(* IEC 61131-3 sources: RL_MAR/experiments/results/ablation/Ablation_random_topo_deepseek-ai_DeepSeek-V3.2_20260603_051006 (part 2) *)

(* ---- med_49.st ---- *)
FUNCTION_BLOCK SmartHVACSystem
VAR_INPUT
    TemperatureSensor : REAL; (* Temperature sensor reading *)
    HumiditySensor : REAL; (* Humidity sensor reading *)
END_VAR

VAR_OUTPUT
    HVACMode : INT := 0; (* HVAC operating mode: 0=Off, 1=Cooling, 2=Heating, 3=Ventilation *)
    HVACFanSpeed : INT := 0; (* Fan speed: 0=Off, 1=Low, 2=Medium, 3=High *)
END_VAR

VAR
    DesiredTemperature : REAL := 24.0; (* Desired temperature setting *)
    DesiredHumidity : REAL := 50.0; (* Desired humidity setting *)
    TemperatureThreshold : REAL := 1.0; (* Temperature tolerance threshold *)
    HumidityThreshold : REAL := 5.0; (* Humidity tolerance threshold *)
    AdjustedHumidity : REAL; (* Sanitized humidity input *)
    AdjustedTemperature : REAL; (* Sanitized temperature input *)
    NeedsVentilation : BOOL; (* Flag for ventilation requirement *)
    NeedsHeating : BOOL; (* Flag for heating requirement *)
    NeedsCooling : BOOL; (* Flag for cooling requirement *)
END_VAR

(* Input Sanitization *)
IF HumiditySensor < 0.0 THEN
    AdjustedHumidity := 0.0;
ELSIF HumiditySensor > 100.0 THEN
    AdjustedHumidity := 100.0;
ELSE
    AdjustedHumidity := HumiditySensor;
END_IF;

IF TemperatureSensor < -50.0 THEN
    AdjustedTemperature := -50.0;
ELSIF TemperatureSensor > 100.0 THEN
    AdjustedTemperature := 100.0;
ELSE
    AdjustedTemperature := TemperatureSensor;
END_IF;

(* Determine System Requirements *)
NeedsVentilation := AdjustedHumidity < (DesiredHumidity - HumidityThreshold);
NeedsHeating := AdjustedTemperature < (DesiredTemperature - TemperatureThreshold);
NeedsCooling := AdjustedTemperature > (DesiredTemperature + TemperatureThreshold);

(* Control Logic with Prioritization *)
IF NeedsHeating THEN
    HVACMode := 2; (* Heating mode *)
    HVACFanSpeed := 3; (* High fan speed *)
ELSIF NeedsCooling THEN
    HVACMode := 1; (* Cooling mode *)
    HVACFanSpeed := 3; (* High fan speed *)
ELSIF NeedsVentilation THEN
    HVACMode := 3; (* Ventilation mode *)
    HVACFanSpeed := 3; (* High fan speed *)
ELSE
    HVACMode := 0; (* Off mode *)
    HVACFanSpeed := 0; (* Fan off *)
END_IF;

END_FUNCTION_BLOCK

(* ---- med_50.st ---- *)
FUNCTION_BLOCK CarParkingSystem
VAR_INPUT
    NewCarSlot : INT; (* Input for new car arrival slot number *)
END_VAR
VAR_OUTPUT
    Elevator1Busy : BOOL; (* Elevator 1 status - busy or idle *)
    Elevator2Busy : BOOL; (* Elevator 2 status - busy or idle *)
    Elevator1Position : INT; (* Elevator 1 current position *)
    Elevator2Position : INT; (* Elevator 2 current position *)
END_VAR
VAR
    Elevator1Target : INT; (* Elevator 1 target floor *)
    Elevator2Target : INT; (* Elevator 2 target floor *)
    CarSlots : ARRAY[1..100] OF BOOL; (* Array to represent parking slots - TRUE if occupied *)
    CurrentSlot : INT; (* Loop counter for scanning slots *)
    bScanComplete : BOOL; (* Flag to indicate slot scanning completion *)
END_VAR

(* Initialize variables *)
IF NOT bScanComplete THEN
    Elevator1Target := 0;
    Elevator2Target := 0;
    Elevator1Position := 0;
    Elevator2Position := 0;
    Elevator1Busy := FALSE;
    Elevator2Busy := FALSE;
    CurrentSlot := 1;
    bScanComplete := TRUE;

    (* Clear all parking slots *)
    FOR CurrentSlot := 1 TO 100 DO
        CarSlots[CurrentSlot] := FALSE;
    END_FOR;
END_IF;

(* Process new car arrival *)
IF NewCarSlot >= 1 AND NewCarSlot <= 100 THEN
    IF NOT CarSlots[NewCarSlot] THEN
        CarSlots[NewCarSlot] := TRUE;

        (* Assign elevator based on slot range *)
        IF NewCarSlot <= 50 THEN
            IF NOT Elevator1Busy THEN
                Elevator1Target := NewCarSlot;
                Elevator1Busy := TRUE;
            END_IF;
        ELSE
            IF NOT Elevator2Busy THEN
                Elevator2Target := NewCarSlot;
                Elevator2Busy := TRUE;
            END_IF;
        END_IF;
    END_IF;
END_IF;

(* Elevator 1 movement logic *)
IF Elevator1Busy THEN
    IF Elevator1Position < Elevator1Target THEN
        Elevator1Position := Elevator1Position + 1;
    ELSIF Elevator1Position > Elevator1Target THEN
        Elevator1Position := Elevator1Position - 1;
    ELSE
        (* Reached target - mark as idle *)
        Elevator1Busy := FALSE;
        Elevator1Target := 0;
    END_IF;
END_IF;

(* Elevator 2 movement logic *)
IF Elevator2Busy THEN
    IF Elevator2Position < Elevator2Target THEN
        Elevator2Position := Elevator2Position + 1;
    ELSIF Elevator2Position > Elevator2Target THEN
        Elevator2Position := Elevator2Position - 1;
    ELSE
        (* Reached target - mark as idle *)
        Elevator2Busy := FALSE;
        Elevator2Target := 0;
    END_IF;
END_IF;

(* Scan for new tasks - only scan when both elevators are idle *)
IF NOT Elevator1Busy AND NOT Elevator2Busy THEN
    FOR CurrentSlot := 1 TO 100 DO
        IF CarSlots[CurrentSlot] THEN
            (* Assign to appropriate elevator *)
            IF CurrentSlot <= 50 THEN
                Elevator1Target := CurrentSlot;
                Elevator1Busy := TRUE;
                EXIT; (* Exit loop after assigning one task *)
            ELSE
                Elevator2Target := CurrentSlot;
                Elevator2Busy := TRUE;
                EXIT; (* Exit loop after assigning one task *)
            END_IF;
        END_IF;
    END_FOR;
END_IF;

END_FUNCTION_BLOCK

(* ---- med_51.st ---- *)
FUNCTION_BLOCK PizzaMakingMachine
VAR_INPUT
    StartButton : BOOL;
    StopButton : BOOL;
    DoughReadySensor : BOOL;
    ToppingsReadySensor : BOOL;
    BakingDoneSensor : BOOL;
END_VAR

VAR_OUTPUT
    DoughRollerMotor : BOOL;
    ToppingDispenser : BOOL;
    ConveyorMotor : BOOL;
    OvenHeater : BOOL;
    OvenTemperature : INT;
END_VAR

VAR
    CurrentState : INT := 0;
    NextState : INT := 0;
END_VAR

(* State Machine Execution *)
CurrentState := NextState;

CASE CurrentState OF
    0: (* IDLE STATE *)
        DoughRollerMotor := FALSE;
        ToppingDispenser := FALSE;
        ConveyorMotor := FALSE;
        OvenHeater := FALSE;
        OvenTemperature := 0;

        IF StartButton AND NOT StopButton THEN
            NextState := 1;
        ELSE
            NextState := 0;
        END_IF;

    1: (* PREPARE_DOUGH STATE *)
        DoughRollerMotor := TRUE;
        ToppingDispenser := FALSE;
        ConveyorMotor := FALSE;
        OvenHeater := FALSE;
        OvenTemperature := 0;

        IF StopButton THEN
            NextState := 0;
        ELSIF DoughReadySensor THEN
            NextState := 2;
        ELSE
            NextState := 1;
        END_IF;

    2: (* ADD_TOPPINGS STATE *)
        DoughRollerMotor := FALSE;
        ToppingDispenser := TRUE;
        ConveyorMotor := FALSE;
        OvenHeater := FALSE;
        OvenTemperature := 0;

        IF StopButton THEN
            NextState := 0;
        ELSIF ToppingsReadySensor THEN
            NextState := 3;
        ELSE
            NextState := 2;
        END_IF;

    3: (* MOVE_TO_OVEN STATE *)
        DoughRollerMotor := FALSE;
        ToppingDispenser := FALSE;
        ConveyorMotor := TRUE;
        OvenHeater := TRUE;
        OvenTemperature := 220;

        IF StopButton THEN
            NextState := 0;
        ELSIF BakingDoneSensor THEN
            NextState := 4;
        ELSE
            NextState := 3;
        END_IF;

    4: (* BAKING_COMPLETE STATE *)
        DoughRollerMotor := FALSE;
        ToppingDispenser := FALSE;
        ConveyorMotor := FALSE;
        OvenHeater := FALSE;
        OvenTemperature := 0;

        IF StopButton OR NOT StartButton THEN
            NextState := 0;
        ELSE
            NextState := 4;
        END_IF;

    ELSE
        (* Error handling: Reset to IDLE state *)
        NextState := 0;
        DoughRollerMotor := FALSE;
        ToppingDispenser := FALSE;
        ConveyorMotor := FALSE;
        OvenHeater := FALSE;
        OvenTemperature := 0;

END_CASE;

END_FUNCTION_BLOCK

(* ---- med_52.st ---- *)
FUNCTION_BLOCK TrafficManagementSystem
VAR_INPUT
    VehicleCount1 : INT;
    VehicleCount2 : INT;
    VehicleCount3 : INT;
    VehicleCount4 : INT;
END_VAR

VAR_OUTPUT
    TrafficLight1 : BOOL;  (* TRUE = Green, FALSE = Red *)
    TrafficLight2 : BOOL;
    TrafficLight3 : BOOL;
    TrafficLight4 : BOOL;
END_VAR

VAR
    tmrPair1 : TON;
    tmrPair2 : TON;
    prevCount1 : INT := 0;
    prevCount2 : INT := 0;
    prevCount3 : INT := 0;
    prevCount4 : INT := 0;
    intendedLight1 : BOOL := FALSE;
    intendedLight2 : BOOL := FALSE;
    intendedLight3 : BOOL := FALSE;
    intendedLight4 : BOOL := FALSE;
    countChangeDetected : BOOL;
END_VAR

(* Detect if any vehicle count has changed since last cycle *)
countChangeDetected := (prevCount1 <> VehicleCount1) OR
                       (prevCount2 <> VehicleCount2) OR
                       (prevCount3 <> VehicleCount3) OR
                       (prevCount4 <> VehicleCount4);

(* Timer for Pair 1 (Intersections 1 & 2) - 5 second minimum green time *)
tmrPair1(
    IN := countChangeDetected,
    PT := T#5s
);

(* Timer for Pair 2 (Intersections 3 & 4) - 5 second minimum green time *)
tmrPair2(
    IN := countChangeDetected,
    PT := T#5s
);

(* Determine intended light states for Pair 1 based on vehicle counts *)
IF VehicleCount1 > VehicleCount2 THEN
    intendedLight1 := TRUE;
    intendedLight2 := FALSE;
ELSIF VehicleCount2 > VehicleCount1 THEN
    intendedLight1 := FALSE;
    intendedLight2 := TRUE;
ELSE
    (* If counts are equal, set both to red for safety *)
    intendedLight1 := FALSE;
    intendedLight2 := FALSE;
END_IF;

(* Determine intended light states for Pair 2 based on vehicle counts *)
IF VehicleCount3 > VehicleCount4 THEN
    intendedLight3 := TRUE;
    intendedLight4 := FALSE;
ELSIF VehicleCount4 > VehicleCount3 THEN
    intendedLight3 := FALSE;
    intendedLight4 := TRUE;
ELSE
    (* If counts are equal, set both to red for safety *)
    intendedLight3 := FALSE;
    intendedLight4 := FALSE;
END_IF;

(* Apply light states with timer logic to prevent rapid toggling *)
(* Pair 1: Only update lights if timer has elapsed or no change detected *)
IF NOT tmrPair1.Q AND countChangeDetected THEN
    (* Hold current states during timer period *)
    TrafficLight1 := TrafficLight1;
    TrafficLight2 := TrafficLight2;
ELSE
    (* Apply intended states when timer elapses *)
    TrafficLight1 := intendedLight1;
    TrafficLight2 := intendedLight2;
END_IF;

(* Pair 2: Only update lights if timer has elapsed or no change detected *)
IF NOT tmrPair2.Q AND countChangeDetected THEN
    (* Hold current states during timer period *)
    TrafficLight3 := TrafficLight3;
    TrafficLight4 := TrafficLight4;
ELSE
    (* Apply intended states when timer elapses *)
    TrafficLight3 := intendedLight3;
    TrafficLight4 := intendedLight4;
END_IF;

(* Update previous counts for next cycle *)
prevCount1 := VehicleCount1;
prevCount2 := VehicleCount2;
prevCount3 := VehicleCount3;
prevCount4 := VehicleCount4;

END_FUNCTION_BLOCK

(* ---- med_53.st ---- *)
FUNCTION_BLOCK PouchMachine
VAR_INPUT
    start_machine: BOOL;
    stop_machine: BOOL;
    EmergencyStop: BOOL;
    HeatingStationReady_1: BOOL;
    HeatingStationReady_2: BOOL;
    HeatingStationReady_3: BOOL;
    HeatingStationReady_4: BOOL;
    HeatingStationReady_5: BOOL;
    HeatingStationReady_6: BOOL;
    HeatingStationReady_7: BOOL;
    HeatingStationReady_8: BOOL;
    CoolingStationReady_1: BOOL;
    CoolingStationReady_2: BOOL;
    CoolingStationReady_3: BOOL;
    CoolingStationReady_4: BOOL;
    CoolingStationReady_5: BOOL;
    CoolingStationReady_6: BOOL;
    CoolingStationReady_7: BOOL;
    CoolingStationReady_8: BOOL;
    Feeder1_TensionOK: BOOL;
    Feeder2_TensionOK: BOOL;
    HorizontalCutterReady: BOOL;
    VerticalCutterReady: BOOL;
END_VAR

VAR_OUTPUT
    machine_ready: BOOL;
    feeder_running: BOOL;
    cutter_running: BOOL;
    heating_running: BOOL;
    cooling_running: BOOL;
    Feeder1_Start: BOOL;
    Feeder2_Start: BOOL;
    HeatingStationStart_1: BOOL;
    HeatingStationStart_2: BOOL;
    HeatingStationStart_3: BOOL;
    HeatingStationStart_4: BOOL;
    HeatingStationStart_5: BOOL;
    HeatingStationStart_6: BOOL;
    HeatingStationStart_7: BOOL;
    HeatingStationStart_8: BOOL;
    CoolingStationStart_1: BOOL;
    CoolingStationStart_2: BOOL;
    CoolingStationStart_3: BOOL;
    CoolingStationStart_4: BOOL;
    CoolingStationStart_5: BOOL;
    CoolingStationStart_6: BOOL;
    CoolingStationStart_7: BOOL;
    CoolingStationStart_8: BOOL;
    HorizontalCutterStart: BOOL;
    VerticalCutterStart: BOOL;
END_VAR

VAR
    startup_complete: BOOL := FALSE;
    shutdown_complete: BOOL := FALSE;
    machine_state: INT := 0;
    startup_timer: TON;
    shutdown_timer: TON;
    heating_stations_ready: BOOL;
    cooling_stations_ready: BOOL;
    tension_established: BOOL;
    cutter_horizontal_ready: BOOL;
    cutter_vertical_ready: BOOL;
    feeder1_ready: BOOL;
    feeder2_ready: BOOL;
    start_rising_edge: R_TRIG;
    stop_rising_edge: R_TRIG;
    emergency_rising_edge: R_TRIG;
    heating_ok_array: ARRAY[1..8] OF BOOL;
    cooling_ok_array: ARRAY[1..8] OF BOOL;
END_VAR

// Edge detection for control signals
start_rising_edge(CLK := start_machine);
stop_rising_edge(CLK := stop_machine);
emergency_rising_edge(CLK := EmergencyStop);

// Initialize status arrays
heating_ok_array[1] := HeatingStationReady_1;
heating_ok_array[2] := HeatingStationReady_2;
heating_ok_array[3] := HeatingStationReady_3;
heating_ok_array[4] := HeatingStationReady_4;
heating_ok_array[5] := HeatingStationReady_5;
heating_ok_array[6] := HeatingStationReady_6;
heating_ok_array[7] := HeatingStationReady_7;
heating_ok_array[8] := HeatingStationReady_8;

cooling_ok_array[1] := CoolingStationReady_1;
cooling_ok_array[2] := CoolingStationReady_2;
cooling_ok_array[3] := CoolingStationReady_3;
cooling_ok_array[4] := CoolingStationReady_4;
cooling_ok_array[5] := CoolingStationReady_5;
cooling_ok_array[6] := CoolingStationReady_6;
cooling_ok_array[7] := CoolingStationReady_7;
cooling_ok_array[8] := CoolingStationReady_8;

// Check all heating stations are ready
heating_stations_ready := heating_ok_array[1] AND heating_ok_array[2] AND
                         heating_ok_array[3] AND heating_ok_array[4] AND
                         heating_ok_array[5] AND heating_ok_array[6] AND
                         heating_ok_array[7] AND heating_ok_array[8];

// Check all cooling stations are ready
cooling_stations_ready := cooling_ok_array[1] AND cooling_ok_array[2] AND
                         cooling_ok_array[3] AND cooling_ok_array[4] AND
                         cooling_ok_array[5] AND cooling_ok_array[6] AND
                         cooling_ok_array[7] AND cooling_ok_array[8];

// Check tension established on both feeders
tension_established := Feeder1_TensionOK AND Feeder2_TensionOK;

// Check both cutters are ready
cutter_horizontal_ready := HorizontalCutterReady;
cutter_vertical_ready := VerticalCutterReady;

// Emergency stop handling - immediate shutdown to state 0
IF EmergencyStop OR emergency_rising_edge.Q THEN
    machine_state := 0;
    startup_timer(IN := FALSE);
    shutdown_timer(IN := FALSE);
END_IF

CASE machine_state OF
    0: // Idle/Stopped state
        machine_ready := FALSE;
        feeder_running := FALSE;
        cutter_running := FALSE;
        heating_running := FALSE;
        cooling_running := FALSE;
        startup_complete := FALSE;
        shutdown_complete := TRUE;

        // Reset all output commands
        Feeder1_Start := FALSE;
        Feeder2_Start := FALSE;
        HorizontalCutterStart := FALSE;
        VerticalCutterStart := FALSE;

        HeatingStationStart_1 := FALSE;
        HeatingStationStart_2 := FALSE;
        HeatingStationStart_3 := FALSE;
        HeatingStationStart_4 := FALSE;
        HeatingStationStart_5 := FALSE;
        HeatingStationStart_6 := FALSE;
        HeatingStationStart_7 := FALSE;
        HeatingStationStart_8 := FALSE;

        CoolingStationStart_1 := FALSE;
        CoolingStationStart_2 := FALSE;
        CoolingStationStart_3 := FALSE;
        CoolingStationStart_4 := FALSE;
        CoolingStationStart_5 := FALSE;
        CoolingStationStart_6 := FALSE;
        CoolingStationStart_7 := FALSE;
        CoolingStationStart_8 := FALSE;

        IF start_rising_edge.Q AND NOT EmergencyStop THEN
            machine_state := 1;
            shutdown_complete := FALSE;
        END_IF;

    1: // Start heating stations
        heating_running := TRUE;

        // Start all heating stations
        HeatingStationStart_1 := TRUE;
        HeatingStationStart_2 := TRUE;
        HeatingStationStart_3 := TRUE;
        HeatingStationStart_4 := TRUE;
        HeatingStationStart_5 := TRUE;
        HeatingStationStart_6 := TRUE;
        HeatingStationStart_7 := TRUE;
        HeatingStationStart_8 := TRUE;

        startup_timer(IN := TRUE, PT := T#5S);
        IF startup_timer.Q AND heating_stations_ready THEN
            machine_state := 2;
            startup_timer(IN := FALSE);
        ELSIF startup_timer.Q AND NOT heating_stations_ready THEN
            // Timeout without all stations ready - go to error state
            machine_state := 99;
        END_IF;

    2: // Start cooling stations
        cooling_running := TRUE;

        // Start all cooling stations
        CoolingStationStart_1 := TRUE;
        CoolingStationStart_2 := TRUE;
        CoolingStationStart_3 := TRUE;
        CoolingStationStart_4 := TRUE;
        CoolingStationStart_5 := TRUE;
        CoolingStationStart_6 := TRUE;
        CoolingStationStart_7 := TRUE;
        CoolingStationStart_8 := TRUE;

        startup_timer(IN := TRUE, PT := T#5S);
        IF startup_timer.Q AND cooling_stations_ready THEN
            machine_state := 3;
            startup_timer(IN := FALSE);
        ELSIF startup_timer.Q AND NOT cooling_stations_ready THEN
            machine_state := 99;
        END_IF;

    3: // Start feeders and establish tension
        feeder_running := TRUE;
        Feeder1_Start := TRUE;
        Feeder2_Start := TRUE;

        startup_timer(IN := TRUE, PT := T#10S);
        IF startup_timer.Q AND tension_established THEN
            feeder1_ready := TRUE;
            feeder2_ready := TRUE;
            machine_state := 4;
            startup_timer(IN := FALSE);
        ELSIF startup_timer.Q AND NOT tension_established THEN
            machine_state := 99;
        END_IF;

    4: // Start cutters
        cutter_running := TRUE;
        HorizontalCutterStart := TRUE;
        VerticalCutterStart := TRUE;

        startup_timer(IN := TRUE, PT := T#3S);
        IF startup_timer.Q AND cutter_horizontal_ready AND cutter_vertical_ready THEN
            machine_state := 5;
            startup_timer(IN := FALSE);
        ELSIF startup_timer.Q AND NOT (cutter_horizontal_ready AND cutter_vertical_ready) THEN
            machine_state := 99;
        END_IF;

    5: // Machine ready state
        machine_ready := TRUE;
        startup_complete := TRUE;

        IF stop_rising_edge.Q OR EmergencyStop THEN
            machine_state := 10;
        END_IF;

    10: // Shutdown - stop cutters
        cutter_running := FALSE;
        HorizontalCutterStart := FALSE;
        VerticalCutterStart := FALSE;

        shutdown_timer(IN := TRUE, PT := T#3S);
        IF shutdown_timer.Q THEN
            machine_state := 11;
            shutdown_timer(IN := FALSE);
        END_IF;

    11: // Shutdown - stop feeders
        feeder_running := FALSE;
        Feeder1_Start := FALSE;
        Feeder2_Start := FALSE;

        shutdown_timer(IN := TRUE, PT := T#5S);
        IF shutdown_timer.Q THEN
            machine_state := 12;
            shutdown_timer(IN := FALSE);
        END_IF;

    12: // Shutdown - stop cooling stations
        cooling_running := FALSE;
        CoolingStationStart_1 := FALSE;
        CoolingStationStart_2 := FALSE;
        CoolingStationStart_3 := FALSE;
        CoolingStationStart_4 := FALSE;
        CoolingStationStart_5 := FALSE;
        CoolingStationStart_6 := FALSE;
        CoolingStationStart_7 := FALSE;
        CoolingStationStart_8 := FALSE;

        shutdown_timer(IN := TRUE, PT := T#5S);
        IF shutdown_timer.Q THEN
            machine_state := 13;
            shutdown_timer(IN := FALSE);
        END_IF;

    13: // Shutdown - stop heating stations
        heating_running := FALSE;
        HeatingStationStart_1 := FALSE;
        HeatingStationStart_2 := FALSE;
        HeatingStationStart_3 := FALSE;
        HeatingStationStart_4 := FALSE;
        HeatingStationStart_5 := FALSE;
        HeatingStationStart_6 := FALSE;
        HeatingStationStart_7 := FALSE;
        HeatingStationStart_8 := FALSE;

        shutdown_timer(IN := TRUE, PT := T#5S);
        IF shutdown_timer.Q THEN
            machine_state := 14;
            shutdown_timer(IN := FALSE);
        END_IF;

    14: // Shutdown complete
        machine_ready := FALSE;
        shutdown_complete := TRUE;

        IF start_rising_edge.Q AND NOT EmergencyStop THEN
            machine_state := 1;
        END_IF;

    99: // Error state
        machine_ready := FALSE;
        feeder_running := FALSE;
        cutter_running := FALSE;
        heating_running := FALSE;
        cooling_running := FALSE;

        // Stop all outputs
        Feeder1_Start := FALSE;
        Feeder2_Start := FALSE;
        HorizontalCutterStart := FALSE;
        VerticalCutterStart := FALSE;

        HeatingStationStart_1 := FALSE;
        HeatingStationStart_2 := FALSE;
        HeatingStationStart_3 := FALSE;
        HeatingStationStart_4 := FALSE;
        HeatingStationStart_5 := FALSE;
        HeatingStationStart_6 := FALSE;
        HeatingStationStart_7 := FALSE;
        HeatingStationStart_8 := FALSE;

        CoolingStationStart_1 := FALSE;
        CoolingStationStart_2 := FALSE;
        CoolingStationStart_3 := FALSE;
        CoolingStationStart_4 := FALSE;
        CoolingStationStart_5 := FALSE;
        CoolingStationStart_6 := FALSE;
        CoolingStationStart_7 := FALSE;
        CoolingStationStart_8 := FALSE;

        // Manual reset required
        IF EmergencyStop THEN
            machine_state := 0;
        END_IF;

    ELSE
        machine_state := 0;
END_CASE;
END_FUNCTION_BLOCK

(* ---- med_54.st ---- *)
FUNCTION_BLOCK FeedForwardControl
VAR_INPUT
    FlowRate1, FlowRate2: REAL; // Input flow rates of reactants
    MixRatio: REAL; // Desired mixing ratio (Reactant1:Reactant2)
END_VAR

VAR_OUTPUT
    OutFlowRate1, OutFlowRate2: REAL; // Output flow rates for reactants to maintain the mixing ratio
END_VAR

VAR
    MixedFlowRate: REAL; // Total mixed flow rate
    LimitedFlowRate1: REAL;
    LimitedFlowRate2: REAL;
    RatioSum: REAL;
END_VAR

// Limit input flow rates to valid range (0 to 100)
LimitedFlowRate1 := LIMIT(0.0, FlowRate1, 100.0);
LimitedFlowRate2 := LIMIT(0.0, FlowRate2, 100.0);

// Calculate total mixed flow rate
MixedFlowRate := LimitedFlowRate1 + LimitedFlowRate2;

// Calculate output flow rates with error handling for division by zero
RatioSum := MixRatio + 1.0;

IF RatioSum <> 0.0 THEN
    // Calculate proportional outputs based on mixing ratio
    OutFlowRate1 := MixedFlowRate * (MixRatio / RatioSum);
    OutFlowRate2 := MixedFlowRate * (1.0 / RatioSum);

    // Limit output flow rates to valid range (0 to 100)
    OutFlowRate1 := LIMIT(0.0, OutFlowRate1, 100.0);
    OutFlowRate2 := LIMIT(0.0, OutFlowRate2, 100.0);
ELSE
    // Handle division by zero case (when MixRatio = -1.0)
    OutFlowRate1 := 0.0;
    OutFlowRate2 := 0.0;
END_IF;

END_FUNCTION_BLOCK

(* ---- med_55.st ---- *)
FUNCTION_BLOCK StateMachineControl
VAR_INPUT
    request : BOOL;
    done : BOOL;
END_VAR

VAR_OUTPUT
    listen : BOOL;
END_VAR

VAR
    state : INT := 0;
END_VAR

CASE state OF
    0: (* Idle state *)
        listen := TRUE;
        IF request THEN
            state := 1;
            listen := FALSE;
        END_IF;

    1: (* Processing state *)
        listen := FALSE;
        IF done THEN
            state := 0;
        END_IF;

    ELSE
        (* Handle unexpected state values *)
        state := 0;
        listen := FALSE;
END_CASE;

END_FUNCTION_BLOCK

(* ---- med_56.st ---- *)
FUNCTION_BLOCK FB_SimpleRepeat
VAR_INPUT
    INPUT_VAR1 : INT := 2;
    INPUT_COUNTER : INT := 4;
END_VAR

VAR_OUTPUT
    OUTPUT_VAR1 : INT;
END_VAR

VAR
    COUNTER : INT;
END_VAR

// Main logic
OUTPUT_VAR1 := INPUT_VAR1;
COUNTER := INPUT_COUNTER;

REPEAT
    OUTPUT_VAR1 := OUTPUT_VAR1 * 2;
    COUNTER := COUNTER - 1;
UNTIL COUNTER = 0
END_REPEAT;

END_FUNCTION_BLOCK

(* ---- med_57.st ---- *)
FUNCTION_BLOCK FB_CourseDifferenceControl
VAR_INPUT
    KOMPASS_GRAD : INT;
    KURS : INT;
END_VAR
VAR_OUTPUT
    KURS_DIFF : INT;
END_VAR
VAR
    iDiff : INT;
END_VAR

IF KOMPASS_GRAD < 0 THEN
    KURS_DIFF := 0;
ELSE
    iDiff := KURS - KOMPASS_GRAD;

    (* Normalize the angular difference to the range [-1800, 1800] *)
    IF iDiff > 1800 THEN
        iDiff := iDiff - 3600;
    ELSIF iDiff < -1800 THEN
        iDiff := iDiff + 3600;
    END_IF;

    KURS_DIFF := iDiff;
END_IF;

END_FUNCTION_BLOCK

(* ---- med_58.st ---- *)
FUNCTION_BLOCK FB_ThresholdAccumulator
VAR_INPUT
    i : INT;
END_VAR

VAR_OUTPUT
    o : INT;
END_VAR

VAR
    s1 : INT;
END_VAR

// Main logic
s1 := 0; // Initialize s1 to 0 at the start of each call

// Process positive input values
IF i > 0 THEN
    s1 := s1 + i;
END_IF;

// Check threshold condition
IF s1 = 42 THEN
    s1 := s1 + 8000;
END_IF;

// Determine final output
IF s1 < 0 THEN
    o := 0;
ELSE
    o := s1;
END_IF;

END_FUNCTION_BLOCK

(* ---- med_59.st ---- *)
FUNCTION_BLOCK FB_ConditionalSelectAndAggregate
VAR_INPUT
    Z : INT;
END_VAR
VAR
    A_X : INT := 42;
    A_Y : INT := 333;
END_VAR
VAR_OUTPUT
    NEW_Z : INT;
END_VAR

IF A_X > Z THEN
    NEW_Z := A_Y;
ELSE
    NEW_Z := Z;
END_IF;
NEW_Z := NEW_Z + A_X + A_Y;
END_FUNCTION_BLOCK

(* ---- med_60.st ---- *)
FUNCTION_BLOCK FB_RequestHandler
VAR_INPUT
    request : BOOL;
    done : BOOL;
END_VAR

VAR_OUTPUT
    listen : BOOL;
END_VAR

VAR
    state : INT := 0;
END_VAR

CASE state OF
    0:
        listen := TRUE;
        IF request THEN
            listen := FALSE;
            state := 1;
        END_IF;

    1:
        listen := FALSE;
        IF done THEN
            listen := TRUE;
            state := 0;
        END_IF;
END_CASE;

END_FUNCTION_BLOCK

(* ---- med_61.st ---- *)
FUNCTION_BLOCK FB_Sum
VAR_INPUT
    maxValue : INT;
END_VAR
VAR_OUTPUT
    wData : WORD;
END_VAR
VAR
    II : INT;
    tempSum : DINT; // Temporary variable for summation
END_VAR

// Initialize
tempSum := 0;
wData := 0;

// Summation loop
FOR II := 0 TO maxValue DO
    tempSum := tempSum + II;
END_FOR

// Assign result with range checking
IF tempSum >= 0 AND tempSum <= 65535 THEN
    wData := WORD(tempSum);
ELSE
    wData := 0; // Handle overflow by resetting to 0
END_IF
END_FUNCTION_BLOCK

(* ---- med_62.st ---- *)
FUNCTION_BLOCK FB_PedestrianTrafficLight
VAR_INPUT
    pedBtnPress : BOOL;
END_VAR
VAR_OUTPUT
    carLightIsGreen : BOOL;
    pedLightIsGreen : BOOL;
    TimeCounter : INT;
END_VAR
VAR
    buttonPressedBefore : BOOL := FALSE;
    CurrentState : INT := 0;
    NextState : INT := 0;
    pedBtnEdge : R_TRIG;
END_VAR

// Edge detection for button press
pedBtnEdge(CLK := pedBtnPress);

// State machine execution
CASE CurrentState OF
    0: // STATE_CAR_GREEN_IDLE
        // Actions executed in this state
        carLightIsGreen := TRUE;
        pedLightIsGreen := FALSE;
        TimeCounter := 0;
        buttonPressedBefore := pedBtnPress;

        // Transition logic from this state
        IF pedBtnEdge.Q AND NOT buttonPressedBefore THEN
            NextState := 1;
        ELSE
            NextState := 0;
        END_IF;

    1: // STATE_CAR_RED_COUNTING
        // Actions executed in this state
        carLightIsGreen := FALSE;
        pedLightIsGreen := FALSE;
        TimeCounter := TimeCounter + 1;

        // Transition logic from this state
        IF TimeCounter >= 10 AND TimeCounter < 40 THEN
            NextState := 2;
        ELSIF TimeCounter >= 40 AND TimeCounter < 50 THEN
            NextState := 3;
        ELSIF TimeCounter >= 50 THEN
            NextState := 0;
        ELSE
            NextState := 1;
        END_IF;

    2: // STATE_PED_GREEN_COUNTING
        // Actions executed in this state
        carLightIsGreen := FALSE;
        pedLightIsGreen := TRUE;
        TimeCounter := TimeCounter + 1;

        // Transition logic from this state
        IF TimeCounter >= 40 AND TimeCounter < 50 THEN
            NextState := 3;
        ELSIF TimeCounter >= 50 THEN
            NextState := 0;
        ELSE
            NextState := 2;
        END_IF;

    3: // STATE_PED_RED_COUNTING
        // Actions executed in this state
        carLightIsGreen := FALSE;
        pedLightIsGreen := FALSE;
        TimeCounter := TimeCounter + 1;

        // Transition logic from this state
        IF TimeCounter >= 50 THEN
            NextState := 0;
        ELSE
            NextState := 3;
        END_IF;
END_CASE;

// State transition
CurrentState := NextState;

END_FUNCTION_BLOCK

(* ---- med_63.st ---- *)
FUNCTION MoveCarToExitGate : BOOL
VAR_INPUT
    SpaceNumber : INT;
END_VAR
// Simulate car movement to exit gate
// In a real system, this would control physical actuators
MoveCarToExitGate := TRUE; // Return TRUE when movement is complete
END_FUNCTION

FUNCTION_BLOCK Automated_Parking_Controller
VAR_INPUT
    EntryGateSensor : BOOL; (* Sensor input for entry gate *)
    ExitGateSensor : BOOL; (* Sensor input for exit gate *)
    CarDetected : BOOL; (* Sensor input for car detection *)
END_VAR
VAR_OUTPUT
    ParkingSpaceNumber : INT := 0; (* Allocated parking space number *)
    RetrievalInProgress : BOOL := FALSE; (* Flag for car retrieval in progress *)
END_VAR
VAR
    ParkingSpaces : ARRAY[1..100] OF BOOL; (* Parking space status: TRUE=Occupied, FALSE=Available *)
    i : INT; (* Loop counter *)
    AssignedSpace : INT := 0; (* Temporary storage for assigned space *)
    RetrievalComplete : BOOL := FALSE; (* Flag to track retrieval completion *)
END_VAR

// Entry Gate Management
IF EntryGateSensor AND NOT RetrievalInProgress THEN
    // Find first available parking space
    AssignedSpace := 0;
    FOR i := 1 TO 100 DO
        IF NOT ParkingSpaces[i] THEN
            AssignedSpace := i;
            EXIT;
        END_IF
    END_FOR

    // If available space found, allocate it
    IF AssignedSpace > 0 THEN
        ParkingSpaces[AssignedSpace] := TRUE;
        ParkingSpaceNumber := AssignedSpace;
    END_IF
END_IF

// Exit Gate Management
IF ExitGateSensor AND (ParkingSpaceNumber > 0) THEN
    // Mark the space as available and reset output
    ParkingSpaces[ParkingSpaceNumber] := FALSE;
    ParkingSpaceNumber := 0;
END_IF

// Car Retrieval Management
IF CarDetected AND NOT RetrievalInProgress AND (ParkingSpaceNumber > 0) THEN
    RetrievalInProgress := TRUE;
    RetrievalComplete := FALSE;
END_IF

IF RetrievalInProgress AND NOT RetrievalComplete THEN
    // Execute car movement to exit gate
    RetrievalComplete := MoveCarToExitGate(ParkingSpaceNumber);

    IF RetrievalComplete THEN
        // Mark space as available and reset
        ParkingSpaces[ParkingSpaceNumber] := FALSE;
        ParkingSpaceNumber := 0;
        RetrievalInProgress := FALSE;
    END_IF
END_IF

END_FUNCTION_BLOCK

(* ---- med_64.st ---- *)
FUNCTION_BLOCK BakeryOvenControl
VAR_INPUT
    TemperatureSensor : REAL;           (* Current oven temperature measurement *)
    HumiditySensor : REAL;              (* Current oven humidity measurement *)
    TemperatureSetpoint : REAL := 180.0; (* Desired temperature setpoint *)
    HumiditySetpoint : REAL := 60.0;    (* Desired humidity setpoint *)
    BakingTimeSetpoint : TIME := T#30m; (* Total baking duration *)
    OvenEnable : BOOL;                  (* Master enable signal for oven operation *)
    TemperatureThreshold : REAL := 2.0; (* Temperature control deadband *)
    HumidityThreshold : REAL := 5.0;    (* Humidity control deadband *)
END_VAR

VAR_OUTPUT
    HeatingElement : BOOL;              (* Control output for heating element *)
    CoolingElement : BOOL;              (* Control output for cooling element *)
    HumidityControl : BOOL;             (* Control output for humidification system *)
    DehumidityControl : BOOL;           (* Control output for dehumidification system *)
    BakingComplete : BOOL;              (* Flag indicating baking cycle completion *)
    RemainingTimeDisplay : TIME;        (* Remaining baking time for display *)
END_VAR

VAR
    RemainingTime : TIME;               (* Internal remaining time counter *)
    OneSecTimer : TON;                  (* Timer for one-second intervals *)
    OvenActive : BOOL;                  (* Internal oven active state *)
    StartBaking : BOOL;                 (* Edge detection for baking start *)
    TemperatureLowLimit : REAL;         (* Calculated temperature lower limit *)
    TemperatureHighLimit : REAL;        (* Calculated temperature upper limit *)
    HumidityLowLimit : REAL;            (* Calculated humidity lower limit *)
    HumidityHighLimit : REAL;           (* Calculated humidity upper limit *)
    PrevOvenEnable : BOOL;              (* Previous state for edge detection *)
END_VAR

(* Calculate control limits based on setpoints and thresholds *)
TemperatureLowLimit := TemperatureSetpoint - TemperatureThreshold;
TemperatureHighLimit := TemperatureSetpoint + TemperatureThreshold;
HumidityLowLimit := HumiditySetpoint - HumidityThreshold;
HumidityHighLimit := HumiditySetpoint + HumidityThreshold;

(* Edge detection for oven enable signal *)
StartBaking := OvenEnable AND NOT PrevOvenEnable;
PrevOvenEnable := OvenEnable;

(* Oven state management *)
IF StartBaking THEN
    (* Initialize baking cycle when oven is first enabled *)
    RemainingTime := BakingTimeSetpoint;
    OvenActive := TRUE;
    BakingComplete := FALSE;
ELSIF NOT OvenEnable THEN
    (* Force oven inactive when enable signal is removed *)
    OvenActive := FALSE;
    BakingComplete := FALSE;
END_IF;

(* Timer logic for one-second decrement *)
OneSecTimer(IN := OvenActive, PT := T#1s);

IF OneSecTimer.Q THEN
    (* Decrement remaining time each second *)
    IF RemainingTime > T#0s THEN
        RemainingTime := RemainingTime - T#1s;
    END_IF;

    (* Check for baking completion *)
    IF RemainingTime <= T#0s THEN
        OvenActive := FALSE;
        BakingComplete := TRUE;
    END_IF;
END_IF;

(* Update display output *)
RemainingTimeDisplay := RemainingTime;

(* Temperature control logic - evaluated every scan *)
IF OvenActive AND (RemainingTime > T#0s) THEN
    (* Heating control *)
    IF TemperatureSensor < TemperatureLowLimit THEN
        HeatingElement := TRUE;
        CoolingElement := FALSE;
    (* Cooling control *)
    ELSIF TemperatureSensor > TemperatureHighLimit THEN
        HeatingElement := FALSE;
        CoolingElement := TRUE;
    (* Within acceptable range *)
    ELSE
        HeatingElement := FALSE;
        CoolingElement := FALSE;
    END_IF;

    (* Humidity control *)
    IF HumiditySensor < HumidityLowLimit THEN
        HumidityControl := TRUE;
        DehumidityControl := FALSE;
    (* Dehumidification control *)
    ELSIF HumiditySensor > HumidityHighLimit THEN
        HumidityControl := FALSE;
        DehumidityControl := TRUE;
    (* Within acceptable range *)
    ELSE
        HumidityControl := FALSE;
        DehumidityControl := FALSE;
    END_IF;
ELSE
    (* Oven inactive or baking complete - force all outputs OFF *)
    HeatingElement := FALSE;
    CoolingElement := FALSE;
    HumidityControl := FALSE;
    DehumidityControl := FALSE;
END_IF;
END_FUNCTION_BLOCK

(* ---- med_65.st ---- *)
FUNCTION_BLOCK TheaterControl
VAR_INPUT
    StartButton : BOOL;        (* Input for starting a performance *)
    StopButton : BOOL;         (* Input for stopping a performance *)
    SceneNumber : INT;         (* Input for selecting the scene or act *)
END_VAR
VAR_OUTPUT
    LightingControl : BOOL;    (* Output for controlling lighting *)
    SoundControl : BOOL;       (* Output for controlling sound *)
    PerformanceInProgress : BOOL; (* Indicator for an ongoing performance *)
END_VAR
VAR
    CurrentState : INT := 0;   (* 0=Idle, 1=Validate Scene, 2=Performance Active *)
    NextState : INT := 0;
END_VAR

(* State machine execution *)
CurrentState := NextState;

CASE CurrentState OF
    0: (* Idle State *)
        LightingControl := FALSE;
        SoundControl := FALSE;
        PerformanceInProgress := FALSE;

        IF StopButton THEN
            NextState := 0;
        ELSIF StartButton AND NOT PerformanceInProgress THEN
            NextState := 1;
        ELSE
            NextState := 0;
        END_IF;

    1: (* Validate Scene State *)
        (* Stop button has highest priority *)
        IF StopButton THEN
            NextState := 0;
        ELSIF (SceneNumber >= 1) AND (SceneNumber <= 3) THEN
            NextState := 2;
        ELSE
            (* Invalid scene number - return to idle *)
            NextState := 0;
        END_IF;

    2: (* Performance Active State *)
        LightingControl := TRUE;
        SoundControl := TRUE;
        PerformanceInProgress := TRUE;

        IF StopButton THEN
            NextState := 0;
        ELSE
            NextState := 2;
        END_IF;

    ELSE
        (* Fallback to idle state for safety *)
        NextState := 0;
END_CASE;

END_FUNCTION_BLOCK

(* ---- med_66.st ---- *)
FUNCTION_BLOCK ElevatorControl
VAR_INPUT
    CurrentPos : INT;
    RequestedPos : INT;
    ButtonPressed : BOOL;
END_VAR

VAR_OUTPUT
    MotorMovingUp : BOOL;
    MotorMovingDown : BOOL;
    DoorIsOpen : BOOL;
END_VAR

VAR
    CurrentState : INT := 0;  (* 0=Idle, 1=MovingUp, 2=MovingDown, 3=Arrived *)
    NextState : INT := 0;
END_VAR

(* State machine implementation *)
CASE CurrentState OF
    0: (* Idle State *)
        (* State actions *)
        MotorMovingUp := FALSE;
        MotorMovingDown := FALSE;
        DoorIsOpen := TRUE;

        (* Transition logic *)
        IF ButtonPressed THEN
            IF RequestedPos > CurrentPos THEN
                NextState := 1;  (* Move up *)
            ELSIF RequestedPos < CurrentPos THEN
                NextState := 2;  (* Move down *)
            ELSE
                NextState := 3;  (* Already at requested floor *)
            END_IF;
        ELSE
            NextState := 0;  (* Remain idle *)
        END_IF;

    1: (* MovingUp State *)
        (* State actions *)
        MotorMovingUp := TRUE;
        MotorMovingDown := FALSE;
        DoorIsOpen := FALSE;

        (* Transition logic *)
        IF CurrentPos = RequestedPos THEN
            NextState := 3;  (* Arrived at target floor *)
        ELSIF RequestedPos < CurrentPos THEN
            NextState := 2;  (* Switch to moving down if new request is below *)
        ELSE
            NextState := 1;  (* Continue moving up *)
        END_IF;

    2: (* MovingDown State *)
        (* State actions *)
        MotorMovingUp := FALSE;
        MotorMovingDown := TRUE;
        DoorIsOpen := FALSE;

        (* Transition logic *)
        IF CurrentPos = RequestedPos THEN
            NextState := 3;  (* Arrived at target floor *)
        ELSIF RequestedPos > CurrentPos THEN
            NextState := 1;  (* Switch to moving up if new request is above *)
        ELSE
            NextState := 2;  (* Continue moving down *)
        END_IF;

    3: (* Arrived State *)
        (* State actions *)
        MotorMovingUp := FALSE;
        MotorMovingDown := FALSE;
        DoorIsOpen := TRUE;

        (* Transition logic *)
        IF ButtonPressed THEN
            IF RequestedPos > CurrentPos THEN
                NextState := 1;  (* Move up *)
            ELSIF RequestedPos < CurrentPos THEN
                NextState := 2;  (* Move down *)
            ELSE
                NextState := 3;  (* Stay arrived *)
            END_IF;
        ELSE
            NextState := 3;  (* Remain arrived *)
        END_IF;

END_CASE;

(* Update state for next cycle *)
CurrentState := NextState;

END_FUNCTION_BLOCK

(* ---- med_67.st ---- *)
FUNCTION_BLOCK FB_FactorialCalculator
VAR_INPUT
    X : INT;
END_VAR

VAR_OUTPUT
    FactorialResult : INT;
    FactorialGoodResult : INT;
END_VAR

VAR
    tempGoodResult : INT;
END_VAR

IF (X >= -3) AND (X <= 3) THEN
    tempGoodResult := X * X * X * X;
    FactorialGoodResult := tempGoodResult;

    IF tempGoodResult > 1 THEN
        FactorialResult := tempGoodResult * (tempGoodResult - 1);
    ELSE
        FactorialResult := tempGoodResult;
    END_IF;
ELSE
    FactorialGoodResult := 0;
    FactorialResult := 1;
END_IF;

END_FUNCTION_BLOCK

(* ---- med_68.st ---- *)
FUNCTION_BLOCK FB_SignalControl
VAR_INPUT
    Int1 : BOOL;
    Int2 : BOOL;
    Int3 : BOOL;
    Int4 : BOOL;
    Int5 : BOOL;
    Int6 : BOOL;
    Int7 : BOOL;
    Int8 : BOOL;
    IntAn1 : UINT;
    IntAn2 : UINT;
    IntAn3 : UINT;
    IntAn4 : UINT;
    IntAn5 : UINT;
    IntAn6 : UINT;
    IntAn7 : UINT;
    IntAn8 : UINT;
    Marca2 : BOOL;  // Input auxiliary control flag
END_VAR

VAR_OUTPUT
    Out1 : BOOL;
    Out2 : BOOL;
    Out3 : BOOL;
    Out4 : BOOL;
    Out5 : BOOL;
    Out6 : BOOL;
    Out7 : BOOL;
    Out8 : BOOL;
    OutAn1 : UINT;
    OutAn2 : UINT;
    OutAn3 : UINT;
    OutAn4 : UINT;
    OutAn5 : UINT;
    OutAn6 : UINT;
    OutAn7 : UINT;
    OutAn8 : UINT;
END_VAR

VAR
    Marca1 : BOOL;  // Internal flag for latching control
    Marca2_Internal : BOOL;  // Internal copy of Marca2 input for logic
END_VAR

// Store input Marca2 in internal variable to avoid overwriting input
Marca2_Internal := Marca2;

// Logic for internal flag Marca1
Marca1 := (NOT Marca2_Internal) AND (Marca1 OR Out1) AND Int1;

// Logic for internal flag Marca2 (using internal copy)
Marca2_Internal := (NOT Marca1) AND (Marca2_Internal OR Out1) AND Int1;

// Latch behavior for Out1
Out1 := (NOT Marca2_Internal) AND (Marca1 OR Out1);

// Direct Boolean pass-through
Out2 := Int2;
Out3 := Int3;
Out4 := Int4;

// Direct unsigned integer pass-through
OutAn1 := IntAn1;
OutAn2 := IntAn2;
OutAn3 := IntAn3;
OutAn4 := IntAn4;

// Conditional outputs for Out5 to Out8
Out5 := (IntAn5 > 1000) AND NOT Int5;
Out6 := (IntAn6 > 1000) AND NOT Int6;
Out7 := (IntAn7 > 1000) AND NOT Int7;
Out8 := (IntAn8 > 1000) AND NOT Int8;

// Pass-through for analog outputs OutAn5 to OutAn8
OutAn5 := IntAn5;
OutAn6 := IntAn6;
OutAn7 := IntAn7;
OutAn8 := IntAn8;

END_FUNCTION_BLOCK

(* ---- med_69.st ---- *)
FUNCTION_BLOCK FB_ValueOut
VAR_INPUT
    valueIn : INT;
    conf : UINT;
END_VAR

VAR_OUTPUT
    ValueOut : INT;
END_VAR

VAR
    tempValue : INT;
END_VAR

METHOD ProcessValue : INT
VAR_INPUT
    inValue : INT;
    inConf : UINT;
END_VAR
VAR
    result : INT;
END_VAR

    result := 0;

    CASE inConf OF
        1, 2:
            IF inValue <> 0 THEN
                result := inValue / 10;
            ELSE
                result := 0;
            END_IF;

        3:
            CASE inValue OF
                0:   result := 0;
                300: result := 163;
                600: result := 331;
            ELSE
                result := 0;
            END_CASE;

        6, 7:
            IF inValue = 100 THEN
                result := 319;
            ELSE
                result := 0;
            END_IF;

    ELSE
        result := 0;
    END_CASE;

    // Ensure non-negative result
    IF result < 0 THEN
        result := 0;
    END_IF;

    ProcessValue := result;
END_METHOD

// Main execution
ValueOut := ProcessValue(valueIn := valueIn, inConf := conf);
END_FUNCTION_BLOCK

(* ---- med_70.st ---- *)
FUNCTION_BLOCK EggIncubatorControl
VAR_INPUT
    StartButton : BOOL;           (* Momentary button to start incubation *)
    StopButton : BOOL;            (* Momentary button to stop incubation *)
    TemperatureSensor : REAL;     (* Current temperature in °C *)
    HumiditySensor : REAL;        (* Current humidity in % *)
END_VAR
VAR_OUTPUT
    HeatingElement : BOOL;        (* Controls heating element *)
    Humidifier : BOOL;            (* Controls humidifier *)
    EggTurningMotor : BOOL;       (* Controls egg turning motor *)
    IncubationInProgress : BOOL;  (* Indicates if incubation is active *)
END_VAR
VAR
    TargetTemperature : REAL;     (* Target temperature setpoint *)
    TargetHumidity : REAL;        (* Target humidity setpoint *)
    TurnIntervalSeconds : INT;    (* Time interval for egg turning *)
    TurnTimerSeconds : INT;       (* Timer for egg turning cycle *)
    TurnMotorState : BOOL;        (* Internal state for motor toggle *)
END_VAR

(* Initialization of parameters *)
TargetTemperature := 37.5;
TargetHumidity := 50.0;
TurnIntervalSeconds := 3600;

(* Main control logic *)
IF StopButton THEN
    (* Emergency/Manual Stop: Reset all outputs and timers *)
    IncubationInProgress := FALSE;
    HeatingElement := FALSE;
    Humidifier := FALSE;
    EggTurningMotor := FALSE;
    TurnTimerSeconds := 0;
    TurnMotorState := FALSE;
ELSIF StartButton AND NOT IncubationInProgress THEN
    (* Start incubation process *)
    IncubationInProgress := TRUE;
    TurnTimerSeconds := 0;
    TurnMotorState := FALSE;
END_IF;

(* Temperature Control - only active when incubation is in progress *)
IF IncubationInProgress THEN
    HeatingElement := TemperatureSensor < TargetTemperature;
ELSE
    HeatingElement := FALSE;
END_IF;

(* Humidity Control - only active when incubation is in progress *)
IF IncubationInProgress THEN
    Humidifier := HumiditySensor < TargetHumidity;
ELSE
    Humidifier := FALSE;
END_IF;

(* Egg Turning Cycle - only active when incubation is in progress *)
IF IncubationInProgress THEN
    (* Increment timer each scan cycle *)
    TurnTimerSeconds := TurnTimerSeconds + 1;

    (* Check if turning interval has been reached *)
    IF TurnTimerSeconds >= TurnIntervalSeconds THEN
        (* Toggle motor state and reset timer *)
        TurnMotorState := NOT TurnMotorState;
        TurnTimerSeconds := 0;
    END_IF;

    (* Output motor state *)
    EggTurningMotor := TurnMotorState;
ELSE
    (* When not in progress, ensure motor is off *)
    EggTurningMotor := FALSE;
    TurnTimerSeconds := 0;
    TurnMotorState := FALSE;
END_IF;

END_FUNCTION_BLOCK

(* ---- med_71.st ---- *)
FUNCTION_BLOCK FB_Fibonacci_Calculator
VAR_INPUT
    N : DINT := 5;
END_VAR
VAR_OUTPUT
    O : DINT := 1;
END_VAR
VAR
    F1 : DINT := 1;
    F2 : DINT := 1;
    CNT : DINT := 2;
    MaxValue : DINT := 32767;
    Temp : DINT;
END_VAR

// Handle edge cases for N <= 2
IF N <= 2 THEN
    O := 1;
    RETURN;
END_IF

// Initialize for N > 2
F1 := 1;
F2 := 1;
CNT := 2;

// Calculate Fibonacci sequence with saturation
WHILE CNT < N DO
    // Check for overflow before calculation
    IF (F1 > (MaxValue - F2)) THEN
        O := MaxValue;
        RETURN;
    END_IF

    Temp := F1 + F2;
    F1 := F2;
    F2 := Temp;
    CNT := CNT + 1;
END_WHILE

O := F2;
END_FUNCTION_BLOCK

PROGRAM Main
VAR
    FibonacciCalc : FB_Fibonacci_Calculator;
    InputValue : DINT := 5;
    Result : DINT;
END_VAR

FibonacciCalc(N := InputValue);
Result := FibonacciCalc.O;
END_PROGRAM

(* ---- med_72.st ---- *)
FUNCTION_BLOCK DigitalSignageManagement
VAR_INPUT
    DisplayLocations : ARRAY[1..10] OF BOOL;    (* Display active status at each location *)
    ContentSource : ARRAY[1..10] OF INT;        (* Requested content for each location *)
END_VAR
VAR_OUTPUT
    CurrentContent : ARRAY[1..10] OF INT;       (* Current displayed content: 1=News, 2=Weather, 3=Promo, 0=None *)
END_VAR
VAR
    i : INT;                                    (* Loop counter *)
END_VAR

(* Main logic: Update content for all locations immediately *)
FOR i := 1 TO 10 DO
    IF DisplayLocations[i] THEN
        (* Display is active - check content source *)
        CASE ContentSource[i] OF
            1: CurrentContent[i] := 1;          (* News *)
            2: CurrentContent[i] := 2;          (* Weather *)
            3: CurrentContent[i] := 3;          (* Promotional Content *)
        ELSE
            CurrentContent[i] := 0;             (* Invalid content code or 0 *)
        END_CASE;
    ELSE
        (* Display is inactive - show no content *)
        CurrentContent[i] := 0;
    END_IF;
END_FOR;

END_FUNCTION_BLOCK

(* ---- med_73.st ---- *)
FUNCTION_BLOCK RoboticWeldingSystem
VAR_INPUT
    RobotArm1Ready : BOOL;    (* Input for robot arm 1 ready status *)
    RobotArm2Ready : BOOL;    (* Input for robot arm 2 ready status *)
    WeldingGunReady : BOOL;   (* Input for welding gun ready status *)
    StartButton : BOOL;       (* Input for start button press *)
    StopButton : BOOL;        (* Input for stop button press *)
END_VAR

VAR_OUTPUT
    WeldingTrigger : BOOL;    (* Output to trigger welding *)
    WeldingComplete : BOOL;   (* Output indicating welding completion *)
END_VAR

VAR
    CurrentState : INT;       (* 0=Idle, 1=Welding, 2=Stopped *)
    AllReady : BOOL;          (* Combined ready status *)
    ReadyLost : BOOL;         (* Flag for lost readiness during welding *)
END_VAR

(* Calculate combined conditions *)
AllReady := RobotArm1Ready AND RobotArm2Ready AND WeldingGunReady;
ReadyLost := NOT AllReady;

(* State machine implementation *)
CASE CurrentState OF
    0: (* Idle State *)
        WeldingTrigger := FALSE;
        WeldingComplete := TRUE;

        IF StopButton THEN
            CurrentState := 2;  (* Go to Stopped state *)
        ELSIF StartButton AND AllReady THEN
            CurrentState := 1;  (* Go to Welding state *)
        ELSE
            CurrentState := 0;  (* Remain in Idle *)
        END_IF;

    1: (* Welding State *)
        WeldingTrigger := TRUE;
        WeldingComplete := FALSE;

        IF StopButton THEN
            CurrentState := 2;  (* Go to Stopped state *)
        ELSIF ReadyLost THEN
            CurrentState := 0;  (* Go to Idle state *)
        ELSE
            CurrentState := 1;  (* Remain in Welding *)
        END_IF;

    2: (* Stopped State *)
        WeldingTrigger := FALSE;
        WeldingComplete := TRUE;

        IF NOT StopButton THEN
            CurrentState := 0;  (* Go to Idle state *)
        ELSE
            CurrentState := 2;  (* Remain in Stopped *)
        END_IF;

    ELSE
        (* Default to Idle state if invalid state *)
        CurrentState := 0;
        WeldingTrigger := FALSE;
        WeldingComplete := TRUE;
END_CASE;

END_FUNCTION_BLOCK

(* ---- med_74.st ---- *)
FUNCTION_BLOCK TrafficManagementSystem
VAR_INPUT
    VehicleCount1 : INT; (* Input for vehicle count at intersection 1 *)
    VehicleCount2 : INT; (* Input for vehicle count at intersection 2 *)
    VehicleCount3 : INT; (* Input for vehicle count at intersection 3 *)
    VehicleCount4 : INT; (* Input for vehicle count at intersection 4 *)
END_VAR
VAR_OUTPUT
    TrafficLight1 : BOOL; (* Output for traffic light at intersection 1 *)
    TrafficLight2 : BOOL; (* Output for traffic light at intersection 2 *)
    TrafficLight3 : BOOL; (* Output for traffic light at intersection 3 *)
    TrafficLight4 : BOOL; (* Output for traffic light at intersection 4 *)
END_VAR

(* Main logic *)
TrafficLight1 := (VehicleCount1 > VehicleCount2);
TrafficLight2 := NOT TrafficLight1;
TrafficLight3 := (VehicleCount3 > VehicleCount4);
TrafficLight4 := NOT TrafficLight3;

END_FUNCTION_BLOCK

(* ---- med_75.st ---- *)
FUNCTION_BLOCK HomeBrewingSystem
VAR_INPUT
    TemperatureSensor : REAL;      (* Current temperature in °C *)
    WaterFlowSensor : REAL;        (* Current water flow in L/min *)
    BrewingStartTime : TIME;       (* Start time of brewing process *)
    BrewingDuration : TIME;        (* Total duration of brewing process *)
END_VAR
VAR_OUTPUT
    HeatingElement : BOOL;         (* Control signal for heating element *)
    AgitationMotor : BOOL;         (* Control signal for agitation motor *)
    HopsDispenser : BOOL;          (* Control signal for hops dispenser *)
    FermentationTank : BOOL;       (* Control signal for fermentation tank transfer *)
END_VAR
VAR
    CurrentTime : TIME;            (* Current system time *)
    ElapsedTime : TIME;            (* Time elapsed since brewing start *)
    ProcessActive : BOOL;          (* Flag indicating if brewing process is active *)
END_VAR

(* Calculate current time and elapsed brewing time *)
CurrentTime := TIME();
ElapsedTime := CurrentTime - BrewingStartTime;

(* Determine if brewing process is within scheduled duration *)
ProcessActive := (ElapsedTime >= T#0s) AND (ElapsedTime <= BrewingDuration);

(* Temperature control: Maintain 65°C *)
IF TemperatureSensor < 65.0 THEN
    HeatingElement := TRUE;
ELSE
    HeatingElement := FALSE;
END_IF;

(* Agitation motor control based on water flow *)
IF WaterFlowSensor > 0.5 THEN
    AgitationMotor := TRUE;
ELSE
    AgitationMotor := FALSE;
END_IF;

(* Hops dispensing after 5 hours, only during active brewing process *)
IF ProcessActive AND (ElapsedTime >= T#5h) THEN
    HopsDispenser := TRUE;
ELSE
    HopsDispenser := FALSE;
END_IF;

(* Fermentation tank transfer after 48 hours, only during active brewing process *)
IF ProcessActive AND (ElapsedTime >= T#48h) THEN
    FermentationTank := TRUE;
ELSE
    FermentationTank := FALSE;
END_IF;

END_FUNCTION_BLOCK

(* ---- med_76.st ---- *)
FUNCTION_BLOCK MultimediaArtInstallationControl
VAR_INPUT
    MotionSensor : BOOL;           (* Motion detection input *)
    AudioTrack : BOOL;             (* Selected audio track *)
    VisualContent : BOOL;          (* Selected visual content *)
    CycleTime : TIME := T#1S;      (* Cycle time for timer increment *)
    MaxDuration : TIME := T#300S;  (* Maximum activation duration *)
END_VAR
VAR_OUTPUT
    LightingControl : BOOL;        (* Lighting control output *)
    AudioControl : BOOL;           (* Audio playback control *)
    VisualControl : BOOL;          (* Visual display control *)
    ActivationTime : TIME;         (* Current activation duration *)
    SystemActive : BOOL;           (* Overall system status *)
END_VAR
VAR
    ActivationTimer : TON;         (* Timer for activation duration *)
    ElapsedTime : TIME;            (* Elapsed activation time *)
    PreviousMotion : BOOL;         (* Previous motion state for edge detection *)
    MotionDetected : BOOL;         (* Rising edge detected motion *)
END_VAR

(* Initialize timer *)
ActivationTimer(IN := MotionSensor, PT := MaxDuration);

(* Detect rising edge of motion *)
MotionDetected := MotionSensor AND NOT PreviousMotion;
PreviousMotion := MotionSensor;

(* Control multimedia elements based on motion detection *)
IF MotionSensor THEN
    (* Activate all elements when motion is detected *)
    LightingControl := TRUE;
    AudioControl := AudioTrack;    (* Only activate if audio track is selected *)
    VisualControl := VisualContent; (* Only activate if visual content is selected *)
    SystemActive := TRUE;

    (* Update elapsed time while motion is detected *)
    IF ActivationTimer.Q THEN
        (* Timer has reached maximum duration *)
        ElapsedTime := MaxDuration;
    ELSE
        (* Calculate elapsed time based on timer's ET output *)
        ElapsedTime := ActivationTimer.ET;
    END_IF;
ELSE
    (* Deactivate all elements when no motion is detected *)
    LightingControl := FALSE;
    AudioControl := FALSE;
    VisualControl := FALSE;
    SystemActive := FALSE;

    (* Reset elapsed time *)
    ElapsedTime := T#0S;

    (* Reset the timer *)
    ActivationTimer(IN := FALSE);
END_IF;

(* Assign output *)
ActivationTime := ElapsedTime;

(* Safety protocol: Power usage monitoring *)
(* This is a placeholder for actual power monitoring logic *)
(* In a real system, you would implement:
   - Current monitoring
   - Temperature sensing
   - Emergency shutdown procedures *)

END_FUNCTION_BLOCK

(* ---- med_77.st ---- *)
FUNCTION_BLOCK OutdoorLEDLightingControl
VAR_INPUT
    AmbientLight : REAL;    (* Ambient light sensor input in Lux *)
    MotionSensor : BOOL;    (* Motion sensor input (TRUE = motion detected) *)
    EnergySaving : BOOL;    (* Energy saving mode switch (TRUE = energy saving ON) *)
END_VAR

VAR_OUTPUT
    Light : BOOL;           (* LED lighting control output (TRUE = lights ON) *)
    EnergyMode : BOOL;      (* Energy saving mode status output *)
END_VAR

(* Main control logic *)
IF MotionSensor THEN
    (* Motion Detection Override: Lights ON, EnergyMode reflects input *)
    Light := TRUE;
ELSE
    (* No motion detected - Ambient Light and Energy Saving Control *)
    IF (AmbientLight < 50.0) AND NOT EnergySaving THEN
        Light := TRUE;
    ELSE
        Light := FALSE;
    END_IF;
END_IF;

(* Energy Mode Status always reflects EnergySaving input *)
EnergyMode := EnergySaving;

END_FUNCTION_BLOCK

(* ---- med_78.st ---- *)
FUNCTION_BLOCK RetractableRoofControl
VAR_INPUT
    RainSensor : BOOL;           (* TRUE if rain is detected *)
    WindSensor : BOOL;           (* TRUE if strong wind is detected *)
    TemperatureSensor : REAL;    (* Current temperature in degrees *)
END_VAR
VAR_OUTPUT
    RoofMotor : BOOL;            (* TRUE = close roof, FALSE = open roof *)
END_VAR

(* Main control logic *)
IF RainSensor AND WindSensor THEN
    (* Highest priority: both rain and strong wind *)
    RoofMotor := TRUE;
ELSIF RainSensor THEN
    (* Second priority: rain only *)
    RoofMotor := TRUE;
ELSIF TemperatureSensor < 20.0 THEN
    (* Third priority: low temperature *)
    RoofMotor := TRUE;
ELSE
    (* Normal conditions: open roof *)
    RoofMotor := FALSE;
END_IF;

END_FUNCTION_BLOCK

(* ---- med_79.st ---- *)
FUNCTION_BLOCK CapsuleFillingMachineControl
VAR_INPUT
    CapsuleWeight : REAL;          (* Current capsule weight *)
    TargetWeight : REAL;           (* Target weight to achieve *)
    CapsuleInPosition : BOOL;      (* Capsule position sensor *)
    HopperEmpty : BOOL;            (* Hopper empty sensor *)
END_VAR

VAR_OUTPUT
    FeederMotor : BOOL;            (* Feeder motor control *)
    FillingMotor : BOOL;           (* Filling motor control *)
    ConveyorMotor : BOOL;          (* Conveyor motor control *)
    FillingInProgress : BOOL;      (* Filling status *)
    ErrorCode : INT;               (* Error code: 0=OK, 1=Capsule timeout, 2=Filling timeout *)
END_VAR

VAR
    // State machine
    CurrentState : INT;            (* 0=IDLE, 1=CONVEYING, 2=FILLING, 3=CONVEYING_OUT *)

    // Timers
    ConveyorTimer : TON;
    FillingTimer : TON;
    ConveyOutTimer : TON;

    // Timing parameters
    ConveyorTime : TIME := T#2S;   (* Time to convey capsule to filling station *)
    MaxFillingTime : TIME := T#10S; (* Maximum allowed filling time *)
    ConveyOutTime : TIME := T#1S;  (* Time to convey filled capsule out *)

    // Control variables
    WeightTolerance : REAL := 0.01; (* 1% tolerance for weight comparison *)
    TargetReached : BOOL;
    FillingStarted : BOOL;

    // Error handling
    CapsuleTimeoutError : BOOL;
    FillingTimeoutError : BOOL;

    // PID-like control variables (simplified proportional control)
    Kp : REAL := 0.8;              (* Proportional gain *)
    PreviousError : REAL;
    ControlOutput : REAL;
    MinMotorSpeed : REAL := 0.1;   (* Minimum motor speed to prevent stalling *)
END_VAR

// Initialize timers
ConveyorTimer(IN:=FALSE, PT:=ConveyorTime);
FillingTimer(IN:=FALSE, PT:=MaxFillingTime);
ConveyOutTimer(IN:=FALSE, PT:=ConveyOutTime);

// Safety Check: Hopper Empty
IF HopperEmpty THEN
    FeederMotor := FALSE;
    FillingMotor := FALSE;
    ConveyorMotor := FALSE;
    FillingInProgress := FALSE;
    CurrentState := 0;  // Return to IDLE state
    ErrorCode := 0;
    RETURN;
END_IF

// Weight Validation: Initial Check
IF CapsuleWeight >= TargetWeight THEN
    FeederMotor := FALSE;
    FillingMotor := FALSE;
    ConveyorMotor := FALSE;
    FillingInProgress := FALSE;
    CurrentState := 0;  // Return to IDLE state
    ErrorCode := 0;
    RETURN;
END_IF

// Calculate if target weight is reached (within tolerance)
TargetReached := (CapsuleWeight >= TargetWeight * (1 - WeightTolerance))
                 AND (CapsuleWeight <= TargetWeight * (1 + WeightTolerance));

// State Machine Implementation
CASE CurrentState OF
    0: (* IDLE State *)
        FeederMotor := FALSE;
        FillingMotor := FALSE;
        ConveyorMotor := FALSE;
        FillingInProgress := FALSE;
        ErrorCode := 0;

        IF CapsuleInPosition THEN
            CurrentState := 1;  // Move to CONVEYING state
            ConveyorTimer(IN:=TRUE);  // Start conveyor timer
        END_IF

    1: (* CONVEYING State *)
        ConveyorMotor := TRUE;
        FillingInProgress := FALSE;

        ConveyorTimer(IN:=TRUE);  // Keep timer running

        IF ConveyorTimer.Q THEN
            // Conveyor timed out without capsule detection
            ConveyorMotor := FALSE;
            CapsuleTimeoutError := TRUE;
            ErrorCode := 1;
            CurrentState := 0;  // Return to IDLE
        ELSIF CapsuleInPosition THEN
            // Capsule successfully conveyed to filling station
            ConveyorTimer(IN:=FALSE);  // Reset timer
            CurrentState := 2;  // Move to FILLING state
            FillingTimer(IN:=TRUE);  // Start filling timer
            FillingStarted := TRUE;
            PreviousError := TargetWeight - CapsuleWeight;  // Initialize error for control
        END_IF

    2: (* FILLING State *)
        ConveyorMotor := FALSE;
        FillingInProgress := TRUE;

        // Simplified proportional control for filling motor
        IF NOT TargetReached AND NOT FillingTimer.Q THEN
            // Calculate error
            VAR
                Error : REAL;
            END_VAR

            Error := TargetWeight - CapsuleWeight;

            // Proportional control with minimum speed
            ControlOutput := Kp * Error;
            IF ControlOutput < MinMotorSpeed THEN
                ControlOutput := MinMotorSpeed;
            ELSIF ControlOutput > 1.0 THEN
                ControlOutput := 1.0;
            END_IF

            // Convert control output to motor command (simplified)
            FillingMotor := TRUE;
            FeederMotor := TRUE;  // Activate feeder to supply material

            PreviousError := Error;
        ELSE
            FillingMotor := FALSE;
            FeederMotor := FALSE;

            IF TargetReached THEN
                // Successful filling
                FillingTimer(IN:=FALSE);  // Reset timer
                CurrentState := 3;  // Move to CONVEYING_OUT state
                ConveyOutTimer(IN:=TRUE);  // Start convey out timer
            ELSIF FillingTimer.Q THEN
                // Filling timeout
                FillingTimeoutError := TRUE;
                ErrorCode := 2;
                CurrentState := 0;  // Return to IDLE
            END_IF
        END_IF

    3: (* CONVEYING_OUT State *)
        FillingMotor := FALSE;
        FeederMotor := FALSE;
        ConveyorMotor := TRUE;
        FillingInProgress := FALSE;

        ConveyOutTimer(IN:=TRUE);  // Keep timer running

        IF ConveyOutTimer.Q THEN
            // Finished conveying out
            ConveyorMotor := FALSE;
            ConveyOutTimer(IN:=FALSE);  // Reset timer
            CurrentState := 0;  // Return to IDLE
        END_IF

END_CASE;

// Reset error flags when returning to IDLE state
IF CurrentState = 0 THEN
    CapsuleTimeoutError := FALSE;
    FillingTimeoutError := FALSE;
END_IF

END_FUNCTION_BLOCK

(* ---- med_80.st ---- *)
FUNCTION_BLOCK DoughMixerControl
VAR_INPUT
    IngredientsDetected : BOOL; (* Input for detecting the presence of ingredients *)
END_VAR

VAR_OUTPUT
    MixingInProgress : BOOL; (* Output for controlling the mixing process - on/off *)
END_VAR

VAR
    MixingTimeElapsed : TIME; (* Timer to track the mixing time *)
    MixingTimeLimit : TIME := T#5S; (* Mixing time limit - 5 seconds *)
    IngredientsDetectedPrev : BOOL; (* Previous state for edge detection *)
    StartTime : TIME; (* Stores the system time when mixing starts *)
    SystemTime : TIME; (* Current system time *)
END_VAR

(* Main logic *)
SystemTime := TIME(); (* Get current system time *)

(* Rising edge detection for IngredientsDetected *)
IF IngredientsDetected AND NOT IngredientsDetectedPrev THEN
    (* Start mixing cycle *)
    MixingInProgress := TRUE;
    StartTime := SystemTime; (* Record start time *)
    MixingTimeElapsed := T#0S; (* Reset elapsed time *)
END_IF;

(* Update previous state for next cycle *)
IngredientsDetectedPrev := IngredientsDetected;

(* Stop conditions *)
IF NOT IngredientsDetected THEN
    (* Stop if ingredients are no longer detected *)
    MixingInProgress := FALSE;
ELSIF MixingInProgress THEN
    (* Calculate elapsed time while mixing *)
    MixingTimeElapsed := SystemTime - StartTime;

    (* Stop if time limit is reached *)
    IF MixingTimeElapsed >= MixingTimeLimit THEN
        MixingInProgress := FALSE;
    END_IF;
END_IF;

(* Ensure timer doesn't increment when not mixing *)
IF NOT MixingInProgress THEN
    MixingTimeElapsed := MixingTimeElapsed; (* Hold current value *)
END_IF;
END_FUNCTION_BLOCK

(* ---- med_81.st ---- *)
FUNCTION_BLOCK SolarPanelTracking
VAR
    PanelAngle : REAL; (* Output for adjusting the solar panel angle *)
    SunriseTime : TIME := T#6H; (* Set the time for sunrise (6:00 AM) *)
    SunsetTime : TIME := T#18H; (* Set the time for sunset (6:00 PM) *)
    NoonTime : TIME := T#12H; (* Set the time for solar noon (12:00 PM) *)
    MorningAngle : REAL := 30.0; (* Set the morning angle for panels *)
    NoonAngle : REAL := 60.0; (* Set the noon angle for panels *)
    EveningAngle : REAL := 30.0; (* Set the evening angle for panels *)
END_VAR
VAR_INPUT
    CurrentTime : TIME;
    SolarIntensity : REAL;
END_VAR

(* Main execution logic *)
IF SolarIntensity >= 90.0 THEN
    (* Solar intensity override - maximum energy capture *)
    PanelAngle := NoonAngle;
ELSE
    (* Time-based tracking logic *)
    IF (CurrentTime < SunriseTime) OR (CurrentTime >= SunsetTime) THEN
        (* Nighttime - panel horizontal *)
        PanelAngle := 0.0;
    ELSIF (CurrentTime >= SunriseTime) AND (CurrentTime < NoonTime) THEN
        (* Morning period *)
        PanelAngle := MorningAngle;
    ELSE
        (* Afternoon/Evening period (NoonTime <= CurrentTime < SunsetTime) *)
        PanelAngle := EveningAngle;
    END_IF;
END_IF;

END_FUNCTION_BLOCK

(* ---- med_82.st ---- *)
FUNCTION_BLOCK PetFeederControl
VAR_INPUT
    CurrentTime : TIME; (* Current system time input *)
END_VAR

VAR_OUTPUT
    FoodDispense : BOOL; (* Food dispenser control signal *)
END_VAR

VAR
    FeedTime1 : TIME := T#8H0M0S; (* First feeding time - 8:00 AM *)
    FeedTime2 : TIME := T#12H0M0S; (* Second feeding time - 12:00 PM *)
    FeedTime3 : TIME := T#18H0M0S; (* Third feeding time - 6:00 PM *)
    FoodAmount : INT := 50; (* Amount of food to dispense in grams - currently unused *)
END_VAR

(* Main dispensing logic *)
FoodDispense := FALSE; (* Default state *)

(* Check if current time is within 30 seconds after FeedTime1 *)
IF (CurrentTime >= FeedTime1) AND (CurrentTime < FeedTime1 + T#30S) THEN
    FoodDispense := TRUE;
END_IF;

(* Check if current time is within 30 seconds after FeedTime2 *)
IF (CurrentTime >= FeedTime2) AND (CurrentTime < FeedTime2 + T#30S) THEN
    FoodDispense := TRUE;
END_IF;

(* Check if current time is within 30 seconds after FeedTime3 *)
IF (CurrentTime >= FeedTime3) AND (CurrentTime < FeedTime3 + T#30S) THEN
    FoodDispense := TRUE;
END_IF;

END_FUNCTION_BLOCK

(* ---- med_83.st ---- *)
FUNCTION_BLOCK AmusementRideControl
VAR_INPUT
    StartButton : BOOL;        (* Start button input *)
    StopButton : BOOL;         (* Emergency stop button input *)
    SpeedSensor : REAL;        (* Speed sensor input (RPM) *)
    SafetySensor : BOOL;       (* Safety sensor status *)
    ResetButton : BOOL;        (* Manual reset button - required after safety trips *)
END_VAR
VAR_OUTPUT
    MotorOn : BOOL := FALSE;   (* Motor control output *)
    BrakeOn : BOOL := TRUE;    (* Brake control output - default fail-safe *)
END_VAR
VAR
    SpeedLimit : REAL := 60.0; (* Maximum allowed speed in RPM *)
    SafetyTrip : BOOL := FALSE;(* Latched safety sensor trip *)
    OverspeedTrip : BOOL := FALSE; (* Latched overspeed trip *)
    EmergencyStopActive : BOOL := FALSE; (* Emergency stop status *)
END_VAR

(* Main safety logic - executed each scan cycle *)
(* HIGHEST PRIORITY: Emergency Stop Handling *)
IF StopButton THEN
    EmergencyStopActive := TRUE;
    MotorOn := FALSE;
    BrakeOn := TRUE;
    (* Emergency stop overrides all other logic *)
    RETURN; (* Exit logic execution for this scan *)
ELSE
    EmergencyStopActive := FALSE;
END_IF;

(* Check for safety violations during operation *)
IF MotorOn THEN
    (* Continuous monitoring while motor is running *)
    IF SpeedSensor > SpeedLimit THEN
        OverspeedTrip := TRUE;
    END_IF;

    IF NOT SafetySensor THEN
        SafetyTrip := TRUE;
    END_IF;
END_IF;

(* Safety Trip Response - Second Highest Priority *)
IF OverspeedTrip OR SafetyTrip THEN
    MotorOn := FALSE;
    BrakeOn := TRUE;
    (* Safety trips require manual reset - do not auto-restart *)
    RETURN; (* Exit logic execution for this scan *)
END_IF;

(* Manual Reset Logic *)
IF ResetButton AND NOT MotorOn THEN
    OverspeedTrip := FALSE;
    SafetyTrip := FALSE;
END_IF;

(* START CONDITION: All conditions must be met simultaneously *)
(* Requires manual reset after any trip *)
IF StartButton
   AND NOT StopButton
   AND (SpeedSensor <= SpeedLimit)
   AND SafetySensor
   AND NOT OverspeedTrip
   AND NOT SafetyTrip
   AND NOT EmergencyStopActive THEN
    (* All start conditions satisfied *)
    MotorOn := TRUE;
    BrakeOn := FALSE;
ELSE
    (* Default fail-safe state *)
    MotorOn := FALSE;
    BrakeOn := TRUE;
END_IF;

END_FUNCTION_BLOCK

(* ---- med_84.st ---- *)
FUNCTION_BLOCK ParcelSortingSystem
VAR_INPUT
    ParcelSizeSensor : REAL;           (* Sensor input for parcel size in mm *)
    DestinationCodeSensor : INT;       (* Destination code: 1=Location A, 2=Location B *)
END_VAR
VAR_OUTPUT
    ConveyorBeltMotor : BOOL;          (* Output for conveyor belt motor: TRUE=On, FALSE=Off *)
    SortingGate1 : BOOL;               (* Output for sorting gate 1: TRUE=Open, FALSE=Closed *)
    SortingGate2 : BOOL;               (* Output for sorting gate 2: TRUE=Open, FALSE=Closed *)
END_VAR
VAR
    SizeThreshold : REAL := 100.0;     (* Threshold to distinguish large vs small parcels *)
    IsLargeParcel : BOOL;              (* Flag indicating parcel is large (>= threshold) *)
    IsSmallParcel : BOOL;              (* Flag indicating parcel is small (< threshold) *)
    IsValidDestination : BOOL;         (* Flag indicating destination code is valid *)
    IsValidSize : BOOL;                (* Flag indicating parcel size is valid *)
END_VAR

(* Initialize outputs to safe default states - all off/closed *)
ConveyorBeltMotor := FALSE;
SortingGate1 := FALSE;
SortingGate2 := FALSE;

(* Validate sensor inputs *)
IsValidSize := (ParcelSizeSensor > 0.0);                    (* Valid size must be positive *)
IsValidDestination := (DestinationCodeSensor = 1) OR (DestinationCodeSensor = 2);  (* Only codes 1 or 2 are valid *)

(* Determine parcel size category based on threshold *)
IsLargeParcel := (ParcelSizeSensor >= SizeThreshold) AND IsValidSize;
IsSmallParcel := (ParcelSizeSensor < SizeThreshold) AND (ParcelSizeSensor > 0.0) AND IsValidSize;

(* Main sorting logic - only execute if both inputs are valid *)
IF IsValidSize AND IsValidDestination THEN
    (* Valid parcel detected - activate conveyor belt *)
    ConveyorBeltMotor := TRUE;

    (* Route parcel based on size and destination *)
    IF IsLargeParcel THEN
        (* Large parcels always go to Sorting Gate 1 regardless of destination *)
        SortingGate1 := TRUE;      (* Open gate 1 *)
        SortingGate2 := FALSE;     (* Ensure gate 2 is closed *)

    ELSIF IsSmallParcel THEN
        (* Small parcels routing depends on destination code *)
        CASE DestinationCodeSensor OF
            1:  (* Destination A - route to Sorting Gate 2 *)
                SortingGate1 := FALSE;     (* Ensure gate 1 is closed *)
                SortingGate2 := TRUE;      (* Open gate 2 *)

            2:  (* Destination B - stay on conveyor, no gates activated *)
                SortingGate1 := FALSE;     (* Ensure gate 1 is closed *)
                SortingGate2 := FALSE;     (* Ensure gate 2 is closed *)
        END_CASE;

    ELSE
        (* Invalid size category - should not reach here due to validation *)
        (* Safety fallback: stop system and close all gates *)
        ConveyorBeltMotor := FALSE;
        SortingGate1 := FALSE;
        SortingGate2 := FALSE;
    END_IF;

ELSE
    (* Invalid input detected - stop system and close all gates *)
    ConveyorBeltMotor := FALSE;
    SortingGate1 := FALSE;
    SortingGate2 := FALSE;
END_IF;

END_FUNCTION_BLOCK

(* ---- med_85.st ---- *)
FUNCTION_BLOCK ShredderControl
VAR_INPUT
    StartButton : BOOL;         (* Momentary start button *)
    StopButton : BOOL;          (* Momentary stop button *)
    EmergencyStop : BOOL;       (* Emergency stop button - active HIGH *)
    MaterialInFeed : BOOL;      (* Material detection sensor *)
    JammedSensor : BOOL;        (* Jam detection sensor - active HIGH *)
END_VAR
VAR_OUTPUT
    MotorControl : BOOL;        (* Motor contactor control *)
    SafetyRelay : BOOL;         (* Safety relay control *)
END_VAR
VAR
    bMotorRunCmd : BOOL;        (* Internal motor run command *)
    bStartEdge : BOOL;          (* Edge detection for start button *)
    bPrevStart : BOOL;          (* Previous start button state *)
    bSafetyOK : BOOL;           (* Combined safety condition *)
END_VAR

(* Edge detection for start button *)
bStartEdge := StartButton AND NOT bPrevStart;
bPrevStart := StartButton;

(* Highest priority safety condition - Emergency Stop OR Jam detected *)
bSafetyOK := NOT EmergencyStop AND NOT JammedSensor;

(* Safety Relay control - active only when safety conditions are met *)
SafetyRelay := bSafetyOK;

(* Normal operation logic - only executed when safety conditions are OK *)
IF bSafetyOK THEN
    (* Start command from button (rising edge) or material feed *)
    IF bStartEdge OR MaterialInFeed THEN
        bMotorRunCmd := TRUE;
    END_IF;

    (* Stop command from stop button *)
    IF StopButton THEN
        bMotorRunCmd := FALSE;
    END_IF;
ELSE
    (* Safety condition violated - force motor stop *)
    bMotorRunCmd := FALSE;
END_IF;

(* Final motor control - requires both run command AND safety OK *)
MotorControl := bMotorRunCmd AND bSafetyOK;

END_FUNCTION_BLOCK

(* ---- med_86.st ---- *)
FUNCTION_BLOCK FruitJuicingBottling
VAR_INPUT
    StartButton : BOOL;     (* Input for starting the process *)
    StopButton : BOOL;      (* Input for stopping the process *)
    FruitSelected : BOOL;   (* Input indicating fruit selection *)
END_VAR
VAR_OUTPUT
    JuiceProcessing : BOOL;     (* Output for controlling juice extraction *)
    BottleFilling : BOOL;       (* Output for controlling bottle filling *)
    CapPlacement : BOOL;        (* Output for placing caps on bottles *)
    Packaging : BOOL;           (* Output for packaging filled bottles *)
    ProcessInProgress : BOOL;   (* Indicator for an ongoing process *)
END_VAR
VAR
    bStartRisingEdge : BOOL;    (* Edge detection for StartButton *)
    bPrevStartButton : BOOL;    (* Previous state of StartButton *)
END_VAR

(* Edge detection for StartButton *)
bStartRisingEdge := StartButton AND NOT bPrevStartButton;
bPrevStartButton := StartButton;

(* Main process control logic *)
IF (bStartRisingEdge AND FruitSelected AND NOT ProcessInProgress) THEN
    ProcessInProgress := TRUE;
END_IF;

IF (StopButton OR NOT FruitSelected) THEN
    ProcessInProgress := FALSE;
END_IF;

(* Concurrent process stage outputs *)
JuiceProcessing := ProcessInProgress;
BottleFilling := ProcessInProgress;
CapPlacement := ProcessInProgress;
Packaging := ProcessInProgress;

END_FUNCTION_BLOCK

(* ---- med_87.st ---- *)
FUNCTION_BLOCK WaterDesalination
VAR_INPUT
    StartButton : BOOL;          (* Input for starting the desalination process *)
    StopButton : BOOL;           (* Input for stopping the desalination process *)
    SalinitySensor : REAL;       (* Input for salinity level measurement *)
END_VAR

VAR_OUTPUT
    SeawaterInletValve : BOOL;       (* Output for seawater inlet valve control *)
    FreshwaterOutletValve : BOOL;    (* Output for freshwater outlet valve control *)
    DesalinationInProgress : BOOL;   (* Indicator for an ongoing desalination process *)
END_VAR

VAR
    MaxSalinity : REAL := 35.0;          (* Maximum allowable salinity in ppm for freshwater *)
    SalinityControlSeconds : INT := 0;   (* Timer for salinity control in seconds *)
    SalinityCheckTimer : TON;            (* Timer for 10-second salinity checks *)
    StartButtonRisingEdge : R_TRIG;      (* Rising edge detector for StartButton *)
    StopButtonRisingEdge : R_TRIG;       (* Rising edge detector for StopButton *)
    SalinityExceeded : BOOL := FALSE;    (* Flag indicating salinity exceeds maximum *)
END_VAR

(* Edge detection for buttons *)
StartButtonRisingEdge(CLK := StartButton);
StopButtonRisingEdge(CLK := StopButton);

(* Main process logic *)
IF StopButton THEN
    (* Immediate stop when StopButton is pressed *)
    DesalinationInProgress := FALSE;
    SeawaterInletValve := FALSE;
    FreshwaterOutletValve := FALSE;
    SalinityControlSeconds := 0;
    SalinityCheckTimer(IN := FALSE, PT := T#10S);
    SalinityExceeded := FALSE;
ELSIF StartButtonRisingEdge.Q AND NOT DesalinationInProgress THEN
    (* Start process when StartButton is pressed and process is not already in progress *)
    DesalinationInProgress := TRUE;
    SeawaterInletValve := TRUE;
    FreshwaterOutletValve := TRUE;
    SalinityControlSeconds := 0;
    SalinityCheckTimer(IN := TRUE, PT := T#10S);
    SalinityExceeded := FALSE;
ELSIF DesalinationInProgress THEN
    (* Process is active - handle salinity monitoring *)
    SeawaterInletValve := TRUE;

    (* 10-second salinity check timer *)
    SalinityCheckTimer(IN := TRUE, PT := T#10S);

    IF SalinityCheckTimer.Q THEN
        (* Timer elapsed - perform salinity check *)
        SalinityControlSeconds := SalinityControlSeconds + 10;
        SalinityCheckTimer(IN := FALSE, PT := T#10S);

        (* Check salinity against maximum *)
        IF SalinitySensor > MaxSalinity THEN
            SalinityExceeded := TRUE;
            FreshwaterOutletValve := FALSE;  (* Close valve if salinity too high *)
        ELSE
            SalinityExceeded := FALSE;
            FreshwaterOutletValve := TRUE;   (* Keep valve open if salinity OK *)
        END_IF;

        (* Restart timer for next check *)
        SalinityCheckTimer(IN := TRUE, PT := T#10S);
    END_IF;

    (* Stop process on rising edge of StopButton *)
    IF StopButtonRisingEdge.Q THEN
        DesalinationInProgress := FALSE;
        SeawaterInletValve := FALSE;
        FreshwaterOutletValve := FALSE;
        SalinityControlSeconds := 0;
        SalinityCheckTimer(IN := FALSE, PT := T#10S);
        SalinityExceeded := FALSE;
    END_IF;
ELSE
    (* Process is idle *)
    DesalinationInProgress := FALSE;
    SeawaterInletValve := FALSE;
    FreshwaterOutletValve := FALSE;
    SalinityCheckTimer(IN := FALSE, PT := T#10S);
END_IF;

END_FUNCTION_BLOCK

(* ---- med_88.st ---- *)
FUNCTION_BLOCK SmartLockerControl
VAR_INPUT
    AccessCode : INT;      (* User entered access code *)
    LockerNumber : INT;    (* Selected locker number (1-10) *)
END_VAR
VAR_OUTPUT
    LockerOpen : BOOL;     (* TRUE when locker should open *)
END_VAR
VAR
    LockerStatus : ARRAY[1..10] OF BOOL;       (* TRUE=locked/occupied, FALSE=empty *)
    LockerAccessCode : ARRAY[1..10] OF INT;    (* Stored access codes *)
    bInitialized : BOOL := FALSE;              (* Initialization flag *)
END_VAR

(* Initialization - runs once on first execution *)
IF NOT bInitialized THEN
    (* Initialize all lockers to TRUE (locked) *)
    LockerStatus[1] := TRUE;
    LockerStatus[2] := TRUE;
    LockerStatus[3] := TRUE;
    LockerStatus[4] := TRUE;
    LockerStatus[5] := TRUE;
    LockerStatus[6] := TRUE;
    LockerStatus[7] := TRUE;
    LockerStatus[8] := TRUE;
    LockerStatus[9] := TRUE;
    LockerStatus[10] := TRUE;

    (* Set predefined access codes *)
    LockerAccessCode[1] := 1234;
    LockerAccessCode[2] := 5678;
    LockerAccessCode[3] := 9876;
    LockerAccessCode[4] := 4321;
    LockerAccessCode[5] := 6543;
    LockerAccessCode[6] := 7890;
    LockerAccessCode[7] := 3456;
    LockerAccessCode[8] := 8765;
    LockerAccessCode[9] := 2345;
    LockerAccessCode[10] := 6789;

    bInitialized := TRUE;
END_IF;

(* Main access control logic *)
LockerOpen := FALSE;  (* Default output state *)

(* Validate locker number range *)
IF (LockerNumber >= 1) AND (LockerNumber <= 10) THEN
    (* Check if access code matches and locker is currently locked *)
    IF (AccessCode = LockerAccessCode[LockerNumber]) AND LockerStatus[LockerNumber] THEN
        LockerOpen := TRUE;                    (* Signal to open the locker *)
        LockerStatus[LockerNumber] := FALSE;   (* Mark locker as empty/unlocked *)
    END_IF;
END_IF;

END_FUNCTION_BLOCK

(* ---- med_89.st ---- *)
FUNCTION_BLOCK SoilTestingDeviceControl
VAR_INPUT
    StartButton : BOOL;           (* Input for starting the testing process *)
    SoilSampleDetected : BOOL;    (* Input for detecting soil sample *)
END_VAR
VAR_OUTPUT
    NutrientPump : BOOL;          (* Output to control nutrient pump *)
    pHAdjustmentPump : BOOL;      (* Output to control pH adjustment pump *)
END_VAR
VAR
    pHSensorValue : REAL;         (* Simulated pH sensor value *)
    NutrientSensorValue : REAL;   (* Simulated nutrient sensor value *)
    TestingStatus : INT;          (* Status: 0=Idle, 1=Testing, 2=Completed *)
    NutrientThreshold : REAL := 0.7;  (* Nutrient level threshold for analysis *)
    pHThreshold : REAL := 6.5;        (* pH level threshold for analysis *)
END_VAR

(* Main logic implementation *)
CASE TestingStatus OF
    0: (* Idle state *)
        (* Initialize sensor values *)
        pHSensorValue := 7.0;
        NutrientSensorValue := 0.5;

        (* Ensure pumps are off *)
        NutrientPump := FALSE;
        pHAdjustmentPump := FALSE;

        (* Transition to Testing state when StartButton is pressed *)
        IF StartButton THEN
            TestingStatus := 1;
            NutrientPump := TRUE;
            pHAdjustmentPump := TRUE;
        END_IF;

    1: (* Testing state *)
        (* Keep pumps active during testing *)
        NutrientPump := TRUE;
        pHAdjustmentPump := TRUE;

        (* Check for sample detection and analysis conditions *)
        IF SoilSampleDetected THEN
            IF (NutrientSensorValue >= NutrientThreshold) AND (pHSensorValue <= pHThreshold) THEN
                TestingStatus := 2;  (* Transition to Completed state *)
                NutrientPump := FALSE;
                pHAdjustmentPump := FALSE;
            END_IF;
        END_IF;

        (* Update simulated sensor values with limits *)
        (* Increment nutrient value with upper limit *)
        NutrientSensorValue := NutrientSensorValue + 0.1;
        IF NutrientSensorValue > 0.9 THEN
            NutrientSensorValue := 0.9;
        END_IF;

        (* Decrement pH value with lower limit *)
        pHSensorValue := pHSensorValue - 0.5;
        IF pHSensorValue < 4.0 THEN
            pHSensorValue := 4.0;
        END_IF;

    2: (* Completed state *)
        (* Ensure pumps are off *)
        NutrientPump := FALSE;
        pHAdjustmentPump := FALSE;

        (* Remain in Completed state - no automatic transition *)

    ELSE
        (* Handle unexpected state values by resetting to Idle *)
        TestingStatus := 0;
END_CASE;

END_FUNCTION_BLOCK

(* ---- med_90.st ---- *)
FUNCTION_BLOCK SushiConveyorControl
VAR_INPUT
    StartButton : BOOL;     (* Input to start the conveyor *)
    StopButton : BOOL;      (* Input to stop the conveyor *)
    EmergencyStop : BOOL;   (* Input for emergency stop *)
END_VAR
VAR_OUTPUT
    ConveyorMotor : BOOL;   (* Output to control the conveyor motor *)
END_VAR
VAR
    BeltRunning : BOOL := FALSE;     (* Status of the conveyor: Running or Stopped *)
    ConveyorTimer : INT := 0;        (* Timer counter for conveyor rotation *)
    RotationTime : INT := 5;         (* Time for one rotation in seconds *)
    TimerPreset : TIME := T#1S;      (* 1 second timer preset for counting *)
    TimerInstance : TON;             (* Timer function block instance *)
END_VAR

(* Emergency Stop - Highest Priority *)
IF EmergencyStop THEN
    ConveyorMotor := FALSE;
    BeltRunning := FALSE;
    ConveyorTimer := 0;
    TimerInstance(IN := FALSE, PT := T#0S);
    RETURN;
END_IF;

(* Start/Stop Control *)
IF StartButton AND NOT BeltRunning THEN
    ConveyorMotor := TRUE;
    BeltRunning := TRUE;
    ConveyorTimer := 0;
    TimerInstance(IN := FALSE, PT := T#0S);
END_IF;

IF StopButton AND BeltRunning THEN
    ConveyorMotor := FALSE;
    BeltRunning := FALSE;
    ConveyorTimer := 0;
    TimerInstance(IN := FALSE, PT := T#0S);
END_IF;

(* Simulated Rotation - Timed On/Off Cycle *)
IF BeltRunning THEN
    (* Start 1-second timer for counting *)
    TimerInstance(IN := TRUE, PT := TimerPreset);

    (* Increment timer every second *)
    IF TimerInstance.Q THEN
        ConveyorTimer := ConveyorTimer + 1;
        TimerInstance(IN := FALSE, PT := T#0S);
    END_IF;

    (* Reset timer when reaching RotationTime *)
    IF ConveyorTimer >= RotationTime THEN
        ConveyorTimer := 0;
    END_IF;

    (* Keep motor ON during entire cycle *)
    ConveyorMotor := TRUE;
ELSE
    (* Ensure motor is OFF when belt is not running *)
    ConveyorMotor := FALSE;
END_IF;

END_FUNCTION_BLOCK

(* ---- med_91.st ---- *)
FUNCTION_BLOCK AGVControlSystem
VAR_INPUT
    MaterialRequest : INT; (* 新的物料请求 *)
END_VAR
VAR_OUTPUT
    AGV1_Ready : BOOL := TRUE; (* AGV 1 就绪状态 *)
    AGV2_Ready : BOOL := TRUE; (* AGV 2 就绪状态 *)
    AGV3_Ready : BOOL := TRUE; (* AGV 3 就绪状态 *)
    SystemErrorCode : INT := 0; (* 系统错误代码 *)
    QueueCount : INT := 0; (* 当前队列任务数 *)
END_VAR
VAR
    (* 队列管理变量 *)
    MaterialQueue : ARRAY[1..10] OF INT; (* 物料处理请求队列 *)
    QueueHead : INT := 1; (* 队列头部指针 *)
    QueueTail : INT := 1; (* 队列尾部指针 *)
    QueueEmpty : BOOL := TRUE; (* 队列空标志 *)
    QueueFull : BOOL := FALSE; (* 队列满标志 *)

    (* AGV状态变量 *)
    AGVStatus : ARRAY[1..3] OF BOOL := [TRUE, TRUE, TRUE]; (* TRUE=就绪, FALSE=工作中 *)
    AGVPosition : ARRAY[1..3] OF INT := [0, 0, 0]; (* AGV当前位置 *)
    AGVTask : ARRAY[1..3] OF INT := [0, 0, 0]; (* AGV当前任务 *)
    AGVTaskProgress : ARRAY[1..3] OF INT := [0, 0, 0]; (* AGV任务进度 *)

    (* 临时变量 *)
    TempRequest : INT;
    TempPosition : INT;
    i : INT;
    j : INT;
    TaskAssigned : BOOL;
    ValidRequest : BOOL;

    (* 状态监控 *)
    SystemIdle : BOOL := TRUE;
    AnyAGVWorking : BOOL := FALSE;
    QueueOverflowError : BOOL := FALSE;
    PositionError : BOOL := FALSE;
    DuplicateTaskError : BOOL := FALSE;
END_VAR

(* 1. 初始化检查和状态重置 *)
IF SystemErrorCode <> 0 THEN
    (* 系统错误时重置状态 *)
    FOR i := 1 TO 3 DO
        AGVStatus[i] := TRUE;
        AGVPosition[i] := 0;
        AGVTask[i] := 0;
        AGVTaskProgress[i] := 0;
    END_FOR;
    QueueHead := 1;
    QueueTail := 1;
    QueueEmpty := TRUE;
    QueueFull := FALSE;
    QueueCount := 0;
    SystemErrorCode := 0;
END_IF;

(* 2. 处理新的物料请求 *)
ValidRequest := (MaterialRequest > 0);
IF ValidRequest THEN
    IF NOT QueueFull THEN
        (* 入队操作 *)
        MaterialQueue[QueueTail] := MaterialRequest;

        (* 更新队列尾部指针 *)
        QueueTail := QueueTail + 1;
        IF QueueTail > 10 THEN
            QueueTail := 1;
        END_IF;

        (* 更新队列状态 *)
        QueueEmpty := FALSE;
        QueueCount := QueueCount + 1;
        IF QueueCount >= 10 THEN
            QueueFull := TRUE;
        END_IF;

        QueueOverflowError := FALSE;
    ELSE
        (* 队列溢出错误 *)
        QueueOverflowError := TRUE;
        SystemErrorCode := 1;
    END_IF;
ELSIF MaterialRequest < 0 THEN
    (* 无效请求错误 *)
    SystemErrorCode := 2;
END_IF;

(* 3. 安全检查：确保AGV位置非负 *)
PositionError := FALSE;
FOR i := 1 TO 3 DO
    IF AGVPosition[i] < 0 THEN
        AGVPosition[i] := 0;
        PositionError := TRUE;
        SystemErrorCode := 3;
    END_IF;
END_FOR;

(* 4. 任务分配：基于优先级AGV1 > AGV2 > AGV3 *)
TaskAssigned := FALSE;
IF (NOT QueueEmpty) AND (SystemErrorCode = 0) THEN
    FOR i := 1 TO 3 DO
        IF (AGVStatus[i] = TRUE) AND (NOT TaskAssigned) THEN
            (* 从队列头部获取任务 *)
            TempRequest := MaterialQueue[QueueHead];

            (* 检查任务是否已被分配 *)
            DuplicateTaskError := FALSE;
            FOR j := 1 TO 3 DO
                IF (j <> i) AND (AGVTask[j] = TempRequest) AND (AGVTask[j] <> 0) THEN
                    DuplicateTaskError := TRUE;
                    SystemErrorCode := 4;
                END_IF;
            END_FOR;

            IF NOT DuplicateTaskError THEN
                (* 分配任务给AGV *)
                AGVTask[i] := TempRequest;
                AGVStatus[i] := FALSE;
                AGVTaskProgress[i] := 0;

                (* 更新队列头部指针 *)
                QueueHead := QueueHead + 1;
                IF QueueHead > 10 THEN
                    QueueHead := 1;
                END_IF;

                (* 更新队列状态 *)
                QueueCount := QueueCount - 1;
                IF QueueCount <= 0 THEN
                    QueueCount := 0;
                    QueueEmpty := TRUE;
                END_IF;
                QueueFull := FALSE;

                TaskAssigned := TRUE;
            END_IF;
        END_IF;
    END_FOR;
END_IF;

(* 5. 模拟AGV任务执行和位置更新 *)
AnyAGVWorking := FALSE;
FOR i := 1 TO 3 DO
    IF AGVStatus[i] = FALSE THEN
        AnyAGVWorking := TRUE;

        IF AGVTask[i] > 0 THEN
            (* 模拟AGV移动 *)
            AGVTaskProgress[i] := AGVTaskProgress[i] + 1;
            AGVPosition[i] := AGVTaskProgress[i];

            (* 检查任务是否完成 *)
            IF AGVTaskProgress[i] >= AGVTask[i] THEN
                (* 任务完成，重置AGV状态 *)
                AGVPosition[i] := 0;
                AGVTask[i] := 0;
                AGVTaskProgress[i] := 0;
                AGVStatus[i] := TRUE;
            END_IF;
        END_IF;
    END_IF;
END_FOR;

(* 6. 更新系统空闲状态 *)
SystemIdle := (QueueEmpty) AND (AGVStatus[1] = TRUE) AND (AGVStatus[2] = TRUE) AND (AGVStatus[3] = TRUE);
IF SystemIdle THEN
    (* 系统空闲时确保所有AGV位置归零 *)
    FOR i := 1 TO 3 DO
        AGVPosition[i] := 0;
    END_FOR;
END_IF;

(* 7. 更新输出状态 *)
AGV1_Ready := AGVStatus[1];
AGV2_Ready := AGVStatus[2];
AGV3_Ready := AGVStatus[3];

(* 8. 资源释放验证 *)
FOR i := 1 TO 3 DO
    IF (AGVStatus[i] = TRUE) AND (AGVTask[i] <> 0) THEN
        (* 状态不一致，强制释放资源 *)
        AGVTask[i] := 0;
        AGVTaskProgress[i] := 0;
        SystemErrorCode := 5;
    END_IF;
END_FOR;

(* 9. 防止重复任务分配（二次检查） *)
FOR i := 1 TO 2 DO
    FOR j := i + 1 TO 3 DO
        IF (AGVTask[i] = AGVTask[j]) AND (AGVTask[i] <> 0) THEN
            (* 发现重复任务，释放较低优先级的AGV *)
            IF j > i THEN
                AGVTask[j] := 0;
                AGVStatus[j] := TRUE;
                AGVTaskProgress[j] := 0;
                AGVPosition[j] := 0;
            END_IF;
            SystemErrorCode := 6;
        END_IF;
    END_FOR;
END_FOR;

(* 10. 状态监控和错误处理汇总 *)
IF SystemErrorCode <> 0 THEN
    (* 有错误时设置所有AGV为就绪状态以确保安全 *)
    AGV1_Ready := TRUE;
    AGV2_Ready := TRUE;
    AGV3_Ready := TRUE;
END_IF;

END_FUNCTION_BLOCK
